C01786=1045.615,121.448,-88.791,170.522,36.741,156.917
C01787=1045.608,121.199,-88.770,170.520,36.740,156.916
C01788=1045.602,120.950,-88.750,170.518,36.739,156.916
C01789=1045.596,120.700,-88.729,170.516,36.737,156.916
C01790=1045.590,120.451,-88.709,170.514,36.736,156.916
C01791=1045.581,120.085,-88.679,170.511,36.733,156.915
C01792=1045.572,119.720,-88.649,170.509,36.731,156.915
C01793=1045.563,119.355,-88.619,170.505,36.729,156.914
C01794=1045.555,118.989,-88.589,170.503,36.726,156.914
C01795=1045.548,118.740,-88.568,170.501,36.725,156.914
C01796=1045.542,118.491,-88.548,170.499,36.723,156.913
C01797=1045.536,118.241,-88.528,170.498,36.722,156.913
C01798=1045.530,117.992,-88.508,170.495,36.721,156.913
C01799=1045.524,117.744,-88.488,170.493,36.719,156.912
C01800=1045.518,117.494,-88.467,170.491,36.718,156.912
C01801=1045.512,117.245,-88.447,170.490,36.716,156.912
C01802=1045.506,116.996,-88.427,170.488,36.715,156.911
C01803=1045.500,116.747,-88.406,170.486,36.713,156.911
C01804=1045.494,116.498,-88.385,170.483,36.711,156.911
C01805=1045.488,116.249,-88.365,170.482,36.710,156.911
C01806=1045.482,116.000,-88.345,170.480,36.708,156.910
C01807=1045.476,115.751,-88.324,170.478,36.707,156.910
C01808=1045.470,115.501,-88.304,170.477,36.705,156.910
C01809=1045.464,115.252,-88.284,170.474,36.703,156.909
C01810=1045.458,115.004,-88.264,170.472,36.702,156.909
C01811=1045.452,114.754,-88.243,170.471,36.700,156.909
C01812=1045.446,114.505,-88.223,170.469,36.699,156.908
C01813=1045.440,114.256,-88.203,170.467,36.698,156.908
C01814=1045.434,114.007,-88.183,170.464,36.696,156.908
C01815=1045.428,113.757,-88.162,170.463,36.695,156.908
C01816=1045.422,113.509,-88.142,170.461,36.693,156.907
C01817=1045.416,113.260,-88.122,170.459,36.692,156.907
C01818=1045.410,113.010,-88.102,170.458,36.690,156.907
C01819=1045.404,112.761,-88.082,170.456,36.689,156.906
C01820=1045.398,112.512,-88.063,170.453,36.687,156.906
C01821=1045.391,112.263,-88.043,170.451,36.686,156.906
C01822=1045.385,112.014,-88.023,170.450,36.684,156.906
C01823=1045.379,111.765,-88.003,170.448,36.683,156.905
C01824=1045.373,111.515,-87.982,170.446,36.681,156.905
C01825=1045.367,111.267,-87.962,170.444,36.680,156.905
C01826=1045.361,111.018,-87.942,170.442,36.679,156.904
C01827=1045.354,110.768,-87.922,170.440,36.677,156.904
C01828=1045.348,110.519,-87.903,170.438,36.676,156.904
C01829=1045.342,110.270,-87.883,170.437,36.674,156.904
C01830=1045.336,110.020,-87.863,170.435,36.673,156.903
C01831=1045.328,109.735,-87.840,170.432,36.671,156.903
C01832=1045.322,109.449,-87.817,170.430,36.669,156.903
C01833=1045.314,109.163,-87.795,170.428,36.668,156.902
C01834=1045.308,108.877,-87.772,170.426,36.666,156.902
C01835=1045.301,108.627,-87.752,170.424,36.665,156.902
C01836=1045.295,108.379,-87.732,170.423,36.664,156.902
C01837=1045.288,108.130,-87.713,170.420,36.662,156.901
C01838=1045.283,107.881,-87.693,170.418,36.661,156.901
C01839=1045.276,107.631,-87.673,170.416,36.659,156.901
C01840=1045.270,107.382,-87.653,170.415,36.658,156.900
C01841=1045.264,107.133,-87.634,170.413,36.656,156.900
C01842=1045.258,106.883,-87.613,170.411,36.655,156.900
C01843=1045.251,106.635,-87.594,170.409,36.653,156.900
C01844=1045.245,106.386,-87.575,170.407,36.652,156.899
C01845=1045.239,106.137,-87.555,170.405,36.651,156.899
C01846=1045.233,105.887,-87.534,170.403,36.650,156.899
C01847=1045.227,105.638,-87.515,170.402,36.648,156.898
C01848=1045.221,105.389,-87.495,170.399,36.646,156.898
C01849=1045.214,105.140,-87.476,170.397,36.645,156.898
C01850=1045.208,104.890,-87.456,170.396,36.643,156.898
C01851=1045.202,104.642,-87.436,170.394,36.642,156.897
C01852=1045.196,104.392,-87.417,170.392,36.641,156.897
C01853=1045.190,104.143,-87.397,170.391,36.639,156.897
C01854=1045.184,103.894,-87.377,170.388,36.638,156.896
C01855=1045.177,103.645,-87.358,170.386,36.637,156.896
C01856=1045.171,103.396,-87.338,170.384,36.635,156.896
C01857=1045.166,103.146,-87.319,170.383,36.633,156.896
C01858=1045.160,102.898,-87.299,170.381,36.632,156.895
C01859=1045.154,102.649,-87.279,170.379,36.630,156.895
C01860=1045.147,102.399,-87.259,170.377,36.629,156.895
C01861=1045.141,102.150,-87.240,170.375,36.628,156.895
C01862=1045.135,101.901,-87.221,170.373,36.626,156.894
C01863=1045.129,101.652,-87.201,170.372,36.625,156.894
C01864=1045.123,101.402,-87.182,170.370,36.624,156.894
C01865=1045.117,101.154,-87.162,170.368,36.622,156.893
C01866=1045.110,100.904,-87.143,170.366,36.620,156.893
C01867=1045.104,100.655,-87.123,170.364,36.619,156.893
C01868=1045.098,100.406,-87.103,170.362,36.618,156.893
C01869=1045.092,100.157,-87.084,170.360,36.616,156.892
C01870=1045.086,99.908,-87.065,170.359,36.615,156.892
C01871=1045.079,99.658,-87.044,170.357,36.614,156.892
C01872=1045.073,99.409,-87.026,170.354,36.612,156.892
C01873=1045.067,99.160,-87.007,170.353,36.611,156.891
C01874=1045.061,98.911,-86.987,170.351,36.609,156.891
C01875=1045.055,98.662,-86.968,170.349,36.608,156.891
C01876=1045.048,98.413,-86.949,170.348,36.607,156.890
C01877=1045.042,98.163,-86.929,170.346,36.605,156.890
C01878=1045.035,97.914,-86.910,170.343,36.604,156.890
C01879=1045.029,97.665,-86.890,170.341,36.602,156.890
C01880=1045.024,97.416,-86.871,170.340,36.601,156.889
C01881=1045.017,97.167,-86.852,170.338,36.600,156.889
C01882=1045.011,96.918,-86.833,170.336,36.599,156.889
C01883=1045.005,96.669,-86.814,170.335,36.597,156.889
C01884=1044.999,96.418,-86.794,170.332,36.596,156.888
C01885=1044.992,96.170,-86.775,170.330,36.594,156.888
C01886=1044.986,95.921,-86.756,170.329,36.593,156.888
C01887=1044.980,95.671,-86.737,170.327,36.591,156.887
C01888=1044.974,95.423,-86.717,170.325,36.590,156.887
C01889=1044.967,95.173,-86.698,170.324,36.589,156.887
C01890=1044.962,94.924,-86.679,170.321,36.587,156.887
C01891=1044.956,94.675,-86.660,170.319,36.586,156.886
C01892=1044.949,94.426,-86.641,170.318,36.584,156.886
C01893=1044.943,94.176,-86.621,170.316,36.583,156.886
C01894=1044.937,93.927,-86.602,170.314,36.582,156.886
C01895=1044.930,93.642,-86.580,170.312,36.580,156.885
C01896=1044.923,93.355,-86.559,170.309,36.579,156.885
C01897=1044.916,93.069,-86.536,170.307,36.577,156.885
C01898=1044.909,92.783,-86.514,170.305,36.575,156.884
C01899=1044.902,92.534,-86.495,170.304,36.574,156.884
C01900=1044.896,92.285,-86.475,170.302,36.572,156.884
C01901=1044.890,92.036,-86.457,170.300,36.571,156.884
C01902=1044.884,91.787,-86.438,170.298,36.569,156.883
C01903=1044.878,91.538,-86.419,170.296,36.568,156.883
C01904=1044.872,91.288,-86.400,170.294,36.567,156.883
C01905=1044.866,91.039,-86.381,170.293,36.566,156.883
C01906=1044.860,90.790,-86.361,170.291,36.564,156.882
C01907=1044.853,90.541,-86.342,170.289,36.562,156.882
C01908=1044.848,90.292,-86.323,170.287,36.561,156.882
C01909=1044.841,90.043,-86.305,170.285,36.560,156.881
C01910=1044.835,89.793,-86.286,170.283,36.559,156.881
C01911=1044.829,89.544,-86.267,170.282,36.557,156.881
C01912=1044.822,89.294,-86.248,170.280,36.556,156.881
C01913=1044.816,89.045,-86.229,170.278,36.554,156.880
C01914=1044.809,88.796,-86.210,170.276,36.553,156.880
C01915=1044.803,88.546,-86.191,170.274,36.552,156.880
C01916=1044.797,88.297,-86.172,170.272,36.551,156.880
C01917=1044.791,88.048,-86.154,170.271,36.549,156.879
C01918=1044.784,87.799,-86.135,170.269,36.548,156.879
C01919=1044.779,87.550,-86.116,170.267,36.546,156.879
C01920=1044.772,87.301,-86.097,170.265,36.545,156.879
C01921=1044.766,87.051,-86.079,170.263,36.544,156.878
C01922=1044.759,86.802,-86.060,170.261,36.543,156.878
C01923=1044.754,86.553,-86.041,170.259,36.541,156.878
C01924=1044.747,86.304,-86.022,170.258,36.540,156.878
C01925=1044.741,86.055,-86.003,170.256,36.538,156.877
C01926=1044.734,85.805,-85.985,170.254,36.537,156.877
C01927=1044.729,85.556,-85.966,170.252,36.536,156.877
C01928=1044.722,85.307,-85.947,170.250,36.534,156.877
C01929=1044.716,85.058,-85.928,170.248,36.533,156.876
C01930=1044.709,84.809,-85.910,170.247,36.532,156.876
C01931=1044.703,84.560,-85.891,170.245,36.530,156.876
C01932=1044.697,84.310,-85.872,170.243,36.529,156.876
C01933=1044.691,84.061,-85.853,170.242,36.528,156.875
C01934=1044.684,83.812,-85.834,170.239,36.526,156.875
C01935=1044.678,83.562,-85.816,170.237,36.525,156.875
C01936=1044.673,83.313,-85.797,170.236,36.524,156.875
C01937=1044.666,83.064,-85.779,170.234,36.522,156.874
C01938=1044.660,82.815,-85.760,170.232,36.521,156.874
C01939=1044.654,82.566,-85.742,170.231,36.519,156.874
C01940=1044.647,82.317,-85.723,170.228,36.518,156.873
C01941=1044.642,82.067,-85.704,170.226,36.517,156.873
C01942=1044.636,81.818,-85.686,170.225,36.516,156.873
C01943=1044.629,81.569,-85.667,170.223,36.514,156.873
C01944=1044.623,81.320,-85.649,170.221,36.513,156.872
C01945=1044.616,81.070,-85.630,170.220,36.511,156.872
C01946=1044.611,80.821,-85.611,170.218,36.510,156.872
C01947=1044.604,80.572,-85.592,170.215,36.509,156.872
C01948=1044.598,80.322,-85.574,170.214,36.507,156.871
C01949=1044.592,80.074,-85.556,170.212,36.506,156.871
C01950=1044.586,79.825,-85.537,170.210,36.504,156.871
C01951=1044.580,79.575,-85.518,170.209,36.503,156.871
C01952=1044.574,79.325,-85.500,170.207,36.502,156.870
C01953=1044.568,79.076,-85.481,170.204,36.500,156.870
C01954=1044.561,78.827,-85.463,170.203,36.499,156.870
C01955=1044.555,78.578,-85.444,170.201,36.497,156.870
C01956=1044.549,78.328,-85.426,170.199,36.496,156.869
C01957=1044.543,78.080,-85.408,170.198,36.495,156.869
C01958=1044.536,77.831,-85.389,170.196,36.494,156.869
C01959=1044.529,77.544,-85.368,170.194,36.492,156.869
C01960=1044.523,77.258,-85.347,170.191,36.491,156.868
C01961=1044.515,76.972,-85.326,170.189,36.489,156.868
C01962=1044.508,76.686,-85.304,170.187,36.487,156.868
C01963=1044.502,76.437,-85.286,170.186,36.486,156.867
C01964=1044.496,76.188,-85.268,170.184,36.485,156.867
C01965=1044.490,75.939,-85.249,170.182,36.484,156.867
C01966=1044.483,75.689,-85.232,170.180,36.482,156.867
C01967=1044.476,75.440,-85.213,170.178,36.481,156.866
C01968=1044.470,75.191,-85.195,170.176,36.479,156.866
C01969=1044.464,74.941,-85.177,170.174,36.478,156.866
C01970=1044.457,74.692,-85.158,170.173,36.477,156.866
C01971=1044.452,74.443,-85.141,170.171,36.476,156.865
C01972=1044.445,74.194,-85.122,170.169,36.474,156.865
C01973=1044.439,73.945,-85.103,170.167,36.473,156.865
C01974=1044.433,73.695,-85.085,170.165,36.472,156.865
C01975=1044.426,73.446,-85.067,170.163,36.471,156.864
C01976=1044.420,73.196,-85.049,170.162,36.469,156.864
C01977=1044.415,72.948,-85.031,170.160,36.467,156.864
C01978=1044.408,72.698,-85.013,170.158,36.466,156.864
C01979=1044.402,72.449,-84.994,170.157,36.465,156.863
C01980=1044.395,72.199,-84.977,170.154,36.464,156.863
C01981=1044.389,71.950,-84.958,170.152,36.462,156.863
C01982=1044.383,71.701,-84.940,170.151,36.461,156.863
C01983=1044.377,71.452,-84.922,170.149,36.460,156.862
C01984=1044.371,71.202,-84.904,170.147,36.459,156.862
C01985=1044.364,70.953,-84.885,170.146,36.457,156.862
C01986=1044.359,70.704,-84.868,170.143,36.455,156.862
C01987=1044.352,70.455,-84.849,170.141,36.454,156.861
C01988=1044.346,70.205,-84.831,170.140,36.453,156.861
C01989=1044.339,69.956,-84.814,170.138,36.452,156.861
C01990=1044.333,69.707,-84.795,170.136,36.450,156.861
C01991=1044.327,69.458,-84.777,170.135,36.449,156.860
C01992=1044.321,69.209,-84.759,170.133,36.448,156.860
C01993=1044.315,68.959,-84.741,170.130,36.447,156.860
C01994=1044.308,68.709,-84.724,170.129,36.445,156.860
C01995=1044.302,68.461,-84.705,170.127,36.444,156.860
C01996=1044.296,68.211,-84.687,170.125,36.443,156.859
C01997=1044.290,67.962,-84.669,170.124,36.442,156.859
C01998=1044.283,67.713,-84.651,170.122,36.440,156.859
C01999=1044.277,67.464,-84.634,170.120,36.438,156.858
C02000=1044.271,67.214,-84.616,170.117,36.437,156.858
C02001=1044.265,66.965,-84.597,170.116,36.436,156.858
C02002=1044.258,66.715,-84.580,170.114,36.435,156.858
C02003=1044.252,66.466,-84.562,170.112,36.433,156.857
C02004=1044.246,66.217,-84.544,170.111,36.432,156.857
C02005=1044.240,65.968,-84.526,170.109,36.431,156.857
C02006=1044.233,65.718,-84.508,170.107,36.430,156.857
C02007=1044.227,65.469,-84.491,170.105,36.428,156.857
C02008=1044.221,65.220,-84.472,170.103,36.427,156.856
C02009=1044.214,64.970,-84.455,170.101,36.426,156.856
C02010=1044.209,64.721,-84.437,170.100,36.425,156.856
C02011=1044.202,64.472,-84.419,170.098,36.423,156.856
C02012=1044.195,64.223,-84.401,170.096,36.422,156.855
C02013=1044.189,63.973,-84.383,170.095,36.421,156.855
C02014=1044.184,63.724,-84.366,170.093,36.420,156.855
C02015=1044.177,63.475,-84.348,170.090,36.418,156.855
C02016=1044.170,63.225,-84.331,170.088,36.417,156.854
C02017=1044.164,62.976,-84.313,170.087,36.416,156.854
C02018=1044.157,62.727,-84.295,170.085,36.415,156.854
C02019=1044.151,62.478,-84.278,170.083,36.413,156.854
C02020=1044.144,62.228,-84.260,170.082,36.412,156.853
C02021=1044.139,61.979,-84.243,170.080,36.411,156.853
C02022=1044.132,61.730,-84.225,170.078,36.410,156.853
C02023=1044.124,61.443,-84.205,170.075,36.408,156.853
C02024=1044.117,61.157,-84.185,170.073,36.407,156.853
C02025=1044.110,60.871,-84.165,170.071,36.406,156.852
C02026=1044.103,60.585,-84.145,170.069,36.404,156.852
C02027=1044.096,60.335,-84.127,170.068,36.403,156.852
C02028=1044.090,60.085,-84.110,170.066,36.402,156.852
C02029=1044.083,59.837,-84.092,170.063,36.401,156.851
C02030=1044.076,59.588,-84.074,170.062,36.399,156.851
C02031=1044.070,59.338,-84.057,170.060,36.398,156.851
C02032=1044.064,59.089,-84.040,170.058,36.397,156.851
C02033=1044.058,58.840,-84.022,170.056,36.396,156.850
C02034=1044.051,58.590,-84.004,170.055,36.394,156.850
C02035=1044.045,58.342,-83.987,170.053,36.393,156.850
C02036=1044.039,58.092,-83.969,170.051,36.392,156.850
C02037=1044.032,57.843,-83.952,170.049,36.391,156.849
C02038=1044.026,57.593,-83.934,170.047,36.389,156.849
C02039=1044.019,57.344,-83.917,170.045,36.388,156.849
C02040=1044.013,57.095,-83.900,170.043,36.387,156.849
C02041=1044.007,56.845,-83.882,170.042,36.386,156.849
C02042=1044.000,56.596,-83.865,170.040,36.385,156.848
C02043=1043.995,56.346,-83.848,170.038,36.384,156.848
C02044=1043.988,56.097,-83.831,170.037,36.382,156.848
C02045=1043.982,55.848,-83.814,170.034,36.381,156.848
C02046=1043.976,55.598,-83.796,170.032,36.380,156.848
C02047=1043.969,55.349,-83.778,170.031,36.379,156.847
C02048=1043.963,55.100,-83.761,170.029,36.377,156.847
C02049=1043.957,54.851,-83.744,170.027,36.376,156.847
C02050=1043.950,54.602,-83.727,170.025,36.375,156.847
C02051=1043.944,54.352,-83.709,170.024,36.373,156.846
C02052=1043.937,54.103,-83.691,170.021,36.372,156.846
C02053=1043.931,53.854,-83.674,170.019,36.371,156.846
C02054=1043.925,53.604,-83.657,170.018,36.370,156.846
C02055=1043.919,53.355,-83.640,170.016,36.368,156.845
C02056=1043.913,53.105,-83.622,170.014,36.367,156.845
C02057=1043.907,52.856,-83.605,170.012,36.366,156.845
C02058=1043.900,52.607,-83.588,170.011,36.365,156.845
C02059=1043.894,52.358,-83.570,170.009,36.363,156.844
C02060=1043.888,52.108,-83.554,170.006,36.362,156.844
C02061=1043.881,51.859,-83.537,170.005,36.361,156.844
C02062=1043.875,51.609,-83.519,170.003,36.360,156.844
C02063=1043.869,51.361,-83.502,170.001,36.358,156.844
C02064=1043.862,51.111,-83.485,170.000,36.357,156.843
C02065=1043.857,50.862,-83.468,169.998,36.356,156.843
C02066=1043.850,50.612,-83.450,169.996,36.355,156.843
C02067=1043.844,50.363,-83.433,169.993,36.353,156.843
C02068=1043.838,50.114,-83.415,169.992,36.352,156.842
C02069=1043.831,49.865,-83.398,169.990,36.351,156.842
C02070=1043.825,49.615,-83.382,169.988,36.349,156.842
C02071=1043.819,49.366,-83.364,169.987,36.348,156.842
C02072=1043.813,49.116,-83.347,169.985,36.347,156.841
C02073=1043.807,48.867,-83.329,169.983,36.346,156.841
C02074=1043.800,48.617,-83.313,169.981,36.344,156.841
C02075=1043.794,48.369,-83.296,169.979,36.343,156.841
C02076=1043.788,48.119,-83.278,169.977,36.342,156.840
C02077=1043.782,47.869,-83.262,169.975,36.341,156.840
C02078=1043.775,47.620,-83.244,169.974,36.339,156.840
C02079=1043.770,47.371,-83.227,169.972,36.338,156.840
C02080=1043.763,47.121,-83.210,169.970,36.337,156.840
C02081=1043.757,46.872,-83.193,169.969,36.336,156.839
C02082=1043.751,46.624,-83.176,169.966,36.334,156.839
C02083=1043.745,46.373,-83.159,169.964,36.333,156.839
C02084=1043.739,46.124,-83.142,169.963,36.332,156.839
C02085=1043.732,45.875,-83.125,169.961,36.330,156.838
C02086=1043.727,45.625,-83.108,169.959,36.329,156.838
C02087=1043.720,45.339,-83.088,169.957,36.328,156.838
C02088=1043.712,45.052,-83.068,169.955,36.326,156.838
C02089=1043.705,44.766,-83.050,169.952,36.325,156.837
C02090=1043.698,44.480,-83.030,169.950,36.323,156.837
C02091=1043.692,44.230,-83.012,169.949,36.322,156.837
C02092=1043.686,43.981,-82.995,169.947,36.321,156.837
C02093=1043.679,43.731,-82.978,169.945,36.320,156.836
C02094=1043.674,43.482,-82.961,169.944,36.318,156.836
C02095=1043.668,43.233,-82.944,169.942,36.317,156.836
C02096=1043.661,42.983,-82.928,169.940,36.316,156.836
C02097=1043.655,42.734,-82.911,169.937,36.315,156.835
C02098=1043.648,42.484,-82.894,169.936,36.313,156.835
C02099=1043.642,42.235,-82.877,169.934,36.312,156.835
C02100=1043.636,41.986,-82.861,169.932,36.311,156.835
C02101=1043.629,41.737,-82.843,169.930,36.309,156.835
C02102=1043.623,41.487,-82.827,169.929,36.308,156.834
C02103=1043.616,41.238,-82.810,169.927,36.307,156.834
C02104=1043.610,40.989,-82.794,169.925,36.306,156.834
C02105=1043.604,40.739,-82.777,169.923,36.305,156.834
C02106=1043.598,40.490,-82.760,169.921,36.304,156.833
C02107=1043.592,40.240,-82.744,169.919,36.302,156.833
C02108=1043.586,39.991,-82.726,169.917,36.301,156.833
C02109=1043.580,39.741,-82.710,169.916,36.300,156.833
C02110=1043.573,39.493,-82.693,169.914,36.299,156.833
C02111=1043.567,39.243,-82.676,169.912,36.297,156.832
C02112=1043.561,38.993,-82.660,169.909,36.296,156.832
C02113=1043.555,38.744,-82.643,169.908,36.295,156.832
C02114=1043.549,38.495,-82.626,169.906,36.294,156.832
C02115=1043.542,38.245,-82.610,169.904,36.293,156.832
C02116=1043.536,37.996,-82.593,169.903,36.292,156.831
C02117=1043.530,37.747,-82.577,169.901,36.290,156.831
C02118=1043.523,37.497,-82.560,169.899,36.289,156.831
C02119=1043.517,37.248,-82.543,169.897,36.288,156.831
C02120=1043.510,36.998,-82.526,169.896,36.287,156.830
C02121=1043.505,36.749,-82.510,169.893,36.285,156.830
C02122=1043.498,36.500,-82.494,169.891,36.285,156.830
C02123=1043.491,36.250,-82.477,169.889,36.283,156.830
C02124=1043.485,36.001,-82.461,169.888,36.282,156.830
C02125=1043.479,35.752,-82.445,169.886,36.281,156.829
C02126=1043.472,35.502,-82.427,169.884,36.280,156.829
C02127=1043.466,35.253,-82.411,169.882,36.279,156.829
C02128=1043.460,35.004,-82.395,169.880,36.278,156.829
C02129=1043.453,34.754,-82.379,169.878,36.276,156.829
C02130=1043.447,34.504,-82.362,169.876,36.275,156.828
C02131=1043.441,34.256,-82.346,169.874,36.274,156.828
C02132=1043.435,34.006,-82.329,169.872,36.273,156.828
C02133=1043.428,33.757,-82.313,169.871,36.272,156.828
C02134=1043.422,33.507,-82.297,169.869,36.271,156.827
C02135=1043.416,33.258,-82.281,169.867,36.269,156.827
C02136=1043.409,33.009,-82.263,169.865,36.268,156.827
C02137=1043.403,32.759,-82.247,169.864,36.267,156.827
C02138=1043.397,32.510,-82.231,169.861,36.266,156.827
C02139=1043.390,32.261,-82.215,169.859,36.265,156.826
C02140=1043.384,32.011,-82.199,169.857,36.264,156.826
C02141=1043.378,31.761,-82.182,169.856,36.262,156.826
C02142=1043.371,31.513,-82.165,169.854,36.261,156.826
C02143=1043.365,31.263,-82.149,169.852,36.260,156.825
C02144=1043.358,31.014,-82.133,169.850,36.259,156.825
C02145=1043.352,30.764,-82.117,169.849,36.258,156.825
C02146=1043.346,30.515,-82.101,169.846,36.257,156.825
C02147=1043.340,30.266,-82.084,169.844,36.255,156.825
C02148=1043.334,30.015,-82.068,169.842,36.254,156.824
C02149=1043.327,29.766,-82.052,169.840,36.253,156.824
C02150=1043.321,29.517,-82.036,169.839,36.252,156.824
C02151=1043.314,29.231,-82.017,169.837,36.251,156.824
C02152=1043.307,28.944,-81.998,169.835,36.249,156.824
C02153=1043.300,28.657,-81.980,169.833,36.248,156.823
C02154=1043.292,28.370,-81.961,169.830,36.246,156.823
C02155=1043.286,28.121,-81.945,169.828,36.245,156.823
C02156=1043.279,27.872,-81.929,169.826,36.244,156.823
C02157=1043.273,27.623,-81.913,169.824,36.243,156.823
C02158=1043.267,27.373,-81.897,169.822,36.242,156.822
C02159=1043.260,27.124,-81.880,169.821,36.241,156.822
C02160=1043.254,26.874,-81.864,169.819,36.240,156.822
C02161=1043.248,26.625,-81.848,169.817,36.239,156.822
C02162=1043.242,26.376,-81.832,169.815,36.237,156.821
C02163=1043.236,26.127,-81.816,169.813,36.236,156.821
C02164=1043.228,25.877,-81.800,169.811,36.236,156.821
C02165=1043.222,25.627,-81.784,169.809,36.234,156.821
C02166=1043.216,25.378,-81.768,169.807,36.233,156.821
C02167=1043.210,25.128,-81.753,169.805,36.232,156.821
C02168=1043.204,24.879,-81.736,169.804,36.231,156.820
C02169=1043.197,24.629,-81.720,169.802,36.230,156.820
C02170=1043.191,24.380,-81.704,169.800,36.228,156.820
C02171=1043.184,24.131,-81.688,169.798,36.228,156.820
C02172=1043.178,23.882,-81.672,169.795,36.227,156.820
C02173=1043.172,23.632,-81.656,169.794,36.225,156.819
C02174=1043.166,23.383,-81.641,169.792,36.224,156.819
C02175=1043.159,23.133,-81.624,169.790,36.223,156.819
C02176=1043.153,22.884,-81.609,169.788,36.222,156.819
C02177=1043.147,22.634,-81.592,169.786,36.221,156.818
C02178=1043.140,22.385,-81.577,169.785,36.219,156.818
C02179=1043.134,22.136,-81.560,169.783,36.219,156.818
C02180=1043.128,21.886,-81.546,169.781,36.218,156.818
C02181=1043.122,21.637,-81.529,169.778,36.216,156.818
C02182=1043.115,21.388,-81.514,169.776,36.215,156.817
C02183=1043.109,21.138,-81.497,169.775,36.214,156.817
C02184=1043.103,20.888,-81.481,169.773,36.213,156.817
C02185=1043.096,20.639,-81.466,169.771,36.212,156.817
C02186=1043.090,20.389,-81.450,169.769,36.211,156.817
C02187=1043.084,20.140,-81.434,169.767,36.210,156.817
C02188=1043.078,19.890,-81.418,169.766,36.209,156.816
C02189=1043.071,19.641,-81.403,169.764,36.207,156.816
C02190=1043.065,19.392,-81.386,169.762,36.207,156.816
C02191=1043.059,19.143,-81.371,169.759,36.205,156.816
C02192=1043.052,18.893,-81.356,169.757,36.204,156.815
C02193=1043.046,18.644,-81.340,169.755,36.203,156.815
C02194=1043.039,18.394,-81.323,169.754,36.202,156.815
C02195=1043.033,18.144,-81.308,169.752,36.201,156.815
C02196=1043.027,17.895,-81.292,169.750,36.200,156.815
C02197=1043.020,17.646,-81.277,169.748,36.199,156.815
C02198=1043.014,17.396,-81.261,169.746,36.198,156.814
C02199=1043.008,17.147,-81.245,169.745,36.197,156.814
C02200=1043.002,16.897,-81.230,169.742,36.196,156.814
C02201=1042.995,16.648,-81.214,169.740,36.194,156.814
C02202=1042.989,16.399,-81.199,169.738,36.194,156.814
C02203=1042.983,16.149,-81.183,169.736,36.193,156.813
C02204=1042.976,15.900,-81.167,169.734,36.191,156.813
C02205=1042.970,15.650,-81.152,169.733,36.190,156.813
C02206=1042.964,15.401,-81.136,169.731,36.189,156.813
C02207=1042.957,15.152,-81.120,169.729,36.188,156.813
C02208=1042.952,14.902,-81.105,169.727,36.187,156.812
C02209=1042.945,14.653,-81.089,169.725,36.186,156.812
C02210=1042.938,14.403,-81.074,169.722,36.185,156.812
C02211=1042.933,14.154,-81.058,169.721,36.184,156.812
C02212=1042.926,13.904,-81.043,169.719,36.183,156.812
C02213=1042.919,13.655,-81.027,169.717,36.182,156.811
C02214=1042.913,13.406,-81.013,169.715,36.181,156.811
C02215=1042.906,13.120,-80.995,169.713,36.180,156.811
C02216=1042.898,12.835,-80.977,169.711,36.178,156.811
C02217=1042.891,12.550,-80.959,169.709,36.177,156.811
C02218=1042.884,12.265,-80.941,169.707,36.176,156.811
C02219=1042.877,12.015,-80.926,169.704,36.175,156.810
C02220=1042.871,11.765,-80.911,169.702,36.174,156.810
C02221=1042.864,11.516,-80.896,169.700,36.173,156.810
C02222=1042.858,11.267,-80.881,169.698,36.172,156.810
C02223=1042.851,11.017,-80.865,169.696,36.171,156.810
C02224=1042.845,10.768,-80.850,169.694,36.170,156.809
C02225=1042.839,10.518,-80.835,169.692,36.169,156.809
C02226=1042.832,10.269,-80.819,169.691,36.168,156.809
C02227=1042.826,10.019,-80.804,169.689,36.167,156.809
C02228=1042.819,9.770,-80.788,169.687,36.166,156.809
C02229=1042.813,9.520,-80.773,169.685,36.165,156.809
C02230=1042.807,9.271,-80.758,169.682,36.164,156.808
C02231=1042.800,9.022,-80.743,169.680,36.163,156.808
C02232=1042.793,8.772,-80.728,169.678,36.162,156.808
C02233=1042.788,8.522,-80.712,169.676,36.161,156.808
C02234=1042.781,8.273,-80.697,169.675,36.160,156.808
C02235=1042.775,8.023,-80.682,169.673,36.159,156.808
C02236=1042.768,7.774,-80.667,169.671,36.158,156.807
C02237=1042.762,7.524,-80.652,169.669,36.157,156.807
C02238=1042.755,7.275,-80.636,169.667,36.156,156.807
C02239=1042.750,7.026,-80.622,169.665,36.155,156.807
C02240=1042.743,6.776,-80.607,169.662,36.154,156.807
C02241=1042.736,6.527,-80.591,169.660,36.153,156.807
C02242=1042.730,6.278,-80.576,169.659,36.152,156.806
C02243=1042.724,6.028,-80.560,169.657,36.151,156.806
C02244=1042.718,5.778,-80.545,169.655,36.150,156.806
C02245=1042.712,5.528,-80.531,169.653,36.149,156.806
C02246=1042.705,5.279,-80.515,169.651,36.148,156.806
C02247=1042.699,5.030,-80.500,169.649,36.147,156.805
C02248=1042.693,4.781,-80.485,169.647,36.146,156.805
C02249=1042.686,4.531,-80.470,169.645,36.145,156.805
C02250=1042.680,4.282,-80.455,169.643,36.144,156.805
C02251=1042.673,4.033,-80.440,169.641,36.143,156.805
C02252=1042.667,3.783,-80.425,169.639,36.142,156.805
C02253=1042.661,3.533,-80.410,169.637,36.141,156.804
C02254=1042.655,3.283,-80.394,169.635,36.140,156.804
C02255=1042.649,3.034,-80.380,169.633,36.139,156.804
C02256=1042.642,2.785,-80.364,169.631,36.138,156.804
C02257=1042.636,2.536,-80.349,169.629,36.137,156.804
C02258=1042.630,2.286,-80.334,169.627,36.136,156.803
C02259=1042.623,2.036,-80.319,169.625,36.135,156.803
C02260=1042.617,1.787,-80.304,169.624,36.134,156.803
C02261=1042.611,1.538,-80.290,169.622,36.133,156.803
C02262=1042.605,1.288,-80.275,169.619,36.132,156.803
C02263=1042.598,1.038,-80.260,169.617,36.131,156.803
C02264=1042.592,0.789,-80.245,169.615,36.130,156.802
C02265=1042.585,0.540,-80.229,169.613,36.129,156.802
C02266=1042.580,0.291,-80.215,169.611,36.128,156.802
C02267=1042.573,0.041,-80.200,169.609,36.127,156.802
C02268=1042.567,-0.209,-80.185,169.607,36.126,156.802
C02269=1042.560,-0.458,-80.170,169.605,36.125,156.802
C02270=1042.555,-0.707,-80.155,169.604,36.124,156.801
C02271=1042.548,-0.957,-80.140,169.602,36.123,156.801
C02272=1042.543,-1.207,-80.125,169.599,36.121,156.801
C02273=1042.536,-1.457,-80.110,169.597,36.121,156.801
C02274=1042.530,-1.705,-80.095,169.595,36.120,156.801
C02275=1042.524,-1.955,-80.080,169.593,36.119,156.801
C02276=1042.518,-2.205,-80.065,169.591,36.118,156.800
C02277=1042.511,-2.454,-80.050,169.589,36.117,156.800
C02278=1042.505,-2.703,-80.036,169.587,36.116,156.800
C02279=1042.498,-2.987,-80.019,169.585,36.114,156.800
C02280=1042.490,-3.270,-80.002,169.583,36.113,156.799
C02281=1042.484,-3.554,-79.985,169.581,36.112,156.799
C02282=1042.477,-3.838,-79.969,169.578,36.111,156.799
C02283=1042.470,-4.087,-79.954,169.576,36.110,156.799
C02284=1042.464,-4.336,-79.940,169.574,36.109,156.799
C02285=1042.458,-4.586,-79.925,169.572,36.108,156.799
C02286=1042.451,-4.835,-79.910,169.570,36.108,156.799
C02287=1042.444,-5.085,-79.896,169.568,36.106,156.798
C02288=1042.439,-5.334,-79.882,169.566,36.106,156.798
C02289=1042.432,-5.584,-79.867,169.564,36.105,156.798
C02290=1042.425,-5.833,-79.852,169.562,36.104,156.798
C02291=1042.419,-6.083,-79.837,169.560,36.103,156.798
C02292=1042.413,-6.332,-79.823,169.558,36.102,156.798
C02293=1042.407,-6.582,-79.808,169.556,36.101,156.797
C02294=1042.400,-6.831,-79.794,169.554,36.101,156.797
C02295=1042.393,-7.081,-79.779,169.551,36.099,156.797
C02296=1042.388,-7.330,-79.765,169.549,36.099,156.797
C02297=1042.381,-7.579,-79.750,169.547,36.097,156.797
C02298=1042.375,-7.830,-79.736,169.545,36.097,156.797
C02299=1042.369,-8.079,-79.722,169.543,36.096,156.797
C02300=1042.362,-8.328,-79.707,169.541,36.095,156.796
C02301=1042.355,-8.578,-79.692,169.539,36.094,156.796
C02302=1042.350,-8.827,-79.678,169.537,36.093,156.796
C02303=1042.343,-9.077,-79.663,169.535,36.092,156.796
C02304=1042.336,-9.326,-79.649,169.533,36.091,156.796
C02305=1042.330,-9.575,-79.635,169.531,36.090,156.796
C02306=1042.324,-9.825,-79.620,169.530,36.090,156.795
C02307=1042.317,-10.075,-79.606,169.527,36.089,156.795
C02308=1042.311,-10.324,-79.591,169.525,36.088,156.795
C02309=1042.305,-10.574,-79.577,169.523,36.087,156.795
C02310=1042.298,-10.823,-79.563,169.521,36.086,156.795
C02311=1042.292,-11.072,-79.548,169.519,36.085,156.795
C02312=1042.286,-11.323,-79.534,169.517,36.084,156.795
C02313=1042.280,-11.571,-79.520,169.515,36.083,156.794
C02314=1042.274,-11.821,-79.505,169.513,36.082,156.794
C02315=1042.267,-12.071,-79.491,169.511,36.082,156.794
C02316=1042.261,-12.320,-79.477,169.509,36.080,156.794
C02317=1042.255,-12.570,-79.463,169.507,36.080,156.794
C02318=1042.248,-12.820,-79.448,169.505,36.079,156.794
C02319=1042.242,-13.068,-79.434,169.502,36.078,156.793
C02320=1042.236,-13.319,-79.419,169.500,36.077,156.793
C02321=1042.230,-13.568,-79.405,169.498,36.076,156.793
C02322=1042.223,-13.818,-79.391,169.496,36.075,156.793
C02323=1042.217,-14.067,-79.377,169.494,36.074,156.793
C02324=1042.211,-14.317,-79.362,169.492,36.073,156.793
C02325=1042.204,-14.566,-79.348,169.490,36.073,156.793
C02326=1042.199,-14.815,-79.334,169.488,36.072,156.792
C02327=1042.192,-15.065,-79.319,169.486,36.071,156.792
C02328=1042.186,-15.314,-79.305,169.484,36.070,156.792
C02329=1042.180,-15.564,-79.291,169.482,36.069,156.792
C02330=1042.173,-15.813,-79.277,169.480,36.068,156.792
C02331=1042.167,-16.063,-79.263,169.478,36.067,156.792
C02332=1042.160,-16.313,-79.249,169.476,36.067,156.792
C02333=1042.155,-16.562,-79.235,169.473,36.066,156.791
C02334=1042.148,-16.812,-79.221,169.471,36.065,156.791
C02335=1042.141,-17.061,-79.207,169.469,36.064,156.791
C02336=1042.135,-17.311,-79.193,169.467,36.063,156.791
C02337=1042.129,-17.560,-79.179,169.465,36.063,156.791
C02338=1042.123,-17.810,-79.165,169.463,36.062,156.791
C02339=1042.116,-18.060,-79.151,169.461,36.061,156.791
C02340=1042.109,-18.309,-79.137,169.459,36.060,156.790
C02341=1042.103,-18.559,-79.123,169.457,36.059,156.790
C02342=1042.097,-18.808,-79.109,169.455,36.059,156.790
C02343=1042.089,-19.090,-79.093,169.452,36.057,156.790
C02344=1042.083,-19.371,-79.078,169.450,36.057,156.790
C02345=1042.075,-19.654,-79.062,169.448,36.056,156.790
C02346=1042.069,-19.936,-79.046,169.444,36.055,156.790
C02347=1042.062,-20.185,-79.032,169.442,36.054,156.789
C02348=1042.055,-20.434,-79.018,169.440,36.053,156.789
C02349=1042.050,-20.684,-79.004,169.438,36.053,156.789
C02350=1042.043,-20.934,-78.990,169.436,36.051,156.789
C02351=1042.036,-21.182,-78.976,169.434,36.051,156.789
C02352=1042.030,-21.433,-78.962,169.432,36.050,156.789
C02353=1042.024,-21.682,-78.949,169.430,36.049,156.789
C02354=1042.018,-21.932,-78.934,169.428,36.049,156.789
C02355=1042.012,-22.181,-78.921,169.426,36.048,156.788
C02356=1042.005,-22.430,-78.907,169.424,36.047,156.788
C02357=1041.999,-22.680,-78.893,169.422,36.046,156.788
C02358=1041.993,-22.929,-78.879,169.420,36.046,156.788
C02359=1041.987,-23.179,-78.865,169.418,36.045,156.788
C02360=1041.980,-23.429,-78.852,169.416,36.044,156.788
C02361=1041.974,-23.679,-78.838,169.413,36.043,156.788
C02362=1041.968,-23.928,-78.824,169.411,36.042,156.788
C02363=1041.962,-24.177,-78.810,169.409,36.042,156.787
C02364=1041.955,-24.427,-78.797,169.407,36.041,156.787
C02365=1041.949,-24.676,-78.783,169.404,36.040,156.787
C02366=1041.942,-24.926,-78.769,169.402,36.039,156.787
C02367=1041.936,-25.176,-78.756,169.400,36.038,156.787
C02368=1041.930,-25.425,-78.741,169.398,36.038,156.787
C02369=1041.924,-25.675,-78.728,169.396,36.036,156.787
C02370=1041.918,-25.924,-78.714,169.394,36.036,156.786
C02371=1041.911,-26.174,-78.700,169.392,36.035,156.786
C02372=1041.905,-26.423,-78.687,169.390,36.034,156.786
C02373=1041.900,-26.673,-78.673,169.388,36.034,156.786
C02374=1041.893,-26.923,-78.659,169.386,36.032,156.786
C02375=1041.887,-27.172,-78.646,169.383,36.032,156.786
C02376=1041.880,-27.422,-78.632,169.381,36.031,156.786
C02377=1041.873,-27.671,-78.618,169.379,36.030,156.786
C02378=1041.867,-27.920,-78.605,169.377,36.030,156.785
C02379=1041.861,-28.170,-78.591,169.374,36.029,156.785
C02380=1041.855,-28.420,-78.578,169.372,36.028,156.785
C02381=1041.849,-28.669,-78.564,169.370,36.028,156.785
C02382=1041.842,-28.919,-78.551,169.368,36.027,156.785
C02383=1041.836,-29.168,-78.537,169.366,36.026,156.785
C02384=1041.829,-29.418,-78.524,169.364,36.026,156.785
C02385=1041.823,-29.667,-78.511,169.362,36.025,156.785
C02386=1041.816,-29.917,-78.497,169.360,36.024,156.785
C02387=1041.810,-30.166,-78.484,169.358,36.024,156.784
C02388=1041.804,-30.416,-78.470,169.355,36.023,156.784
C02389=1041.798,-30.666,-78.457,169.353,36.022,156.784
C02390=1041.791,-30.916,-78.444,169.351,36.022,156.784
C02391=1041.785,-31.165,-78.430,169.349,36.021,156.784
C02392=1041.779,-31.414,-78.417,169.347,36.020,156.784
C02393=1041.772,-31.664,-78.403,169.344,36.020,156.784
C02394=1041.766,-31.914,-78.390,169.342,36.019,156.784
C02395=1041.760,-32.163,-78.377,169.340,36.018,156.784
C02396=1041.753,-32.413,-78.363,169.338,36.018,156.783
C02397=1041.747,-32.662,-78.350,169.335,36.017,156.783
C02398=1041.740,-32.911,-78.337,169.333,36.016,156.783
C02399=1041.734,-33.161,-78.323,169.331,36.015,156.783
C02400=1041.728,-33.412,-78.310,169.329,36.014,156.783
C02401=1041.722,-33.661,-78.297,169.327,36.014,156.783
C02402=1041.716,-33.910,-78.283,169.325,36.013,156.783
C02403=1041.709,-34.160,-78.270,169.323,36.012,156.783
C02404=1041.703,-34.409,-78.257,169.321,36.012,156.782
C02405=1041.697,-34.659,-78.243,169.318,36.011,156.782
C02406=1041.691,-34.909,-78.231,169.316,36.010,156.782
C02407=1041.683,-35.189,-78.216,169.314,36.010,156.782
C02408=1041.677,-35.471,-78.201,169.312,36.009,156.782
C02409=1041.669,-35.751,-78.186,169.309,36.008,156.782
C02410=1041.663,-36.033,-78.171,169.306,36.008,156.782
C02411=1041.657,-36.282,-78.157,169.304,36.007,156.782
C02412=1041.650,-36.531,-78.144,169.301,36.006,156.782
C02413=1041.644,-36.781,-78.131,169.299,36.006,156.782
C02414=1041.637,-37.031,-78.117,169.297,36.005,156.781
C02415=1041.632,-37.280,-78.105,169.295,36.004,156.781
C02416=1041.625,-37.530,-78.091,169.293,36.004,156.781
C02417=1041.619,-37.779,-78.078,169.291,36.003,156.781
C02418=1041.613,-38.030,-78.065,169.289,36.002,156.781
C02419=1041.606,-38.279,-78.052,169.287,36.002,156.781
C02420=1041.600,-38.528,-78.039,169.284,36.001,156.781
C02421=1041.594,-38.778,-78.026,169.282,36.000,156.781
C02422=1041.588,-39.027,-78.013,169.280,36.000,156.781
C02423=1041.581,-39.277,-77.999,169.278,35.999,156.780
C02424=1041.575,-39.527,-77.987,169.276,35.998,156.780
C02425=1041.568,-39.776,-77.974,169.274,35.998,156.780
C02426=1041.562,-40.025,-77.961,169.271,35.997,156.780
C02427=1041.556,-40.275,-77.948,169.269,35.997,156.780
C02428=1041.549,-40.525,-77.935,169.267,35.996,156.780
C02429=1041.543,-40.775,-77.923,169.265,35.996,156.780
C02430=1041.537,-41.024,-77.909,169.262,35.995,156.780
C02431=1041.530,-41.273,-77.896,169.259,35.994,156.780
C02432=1041.524,-41.523,-77.884,169.257,35.994,156.780
C02433=1041.518,-41.772,-77.870,169.255,35.993,156.780
C02434=1041.511,-42.023,-77.858,169.253,35.993,156.780
C02435=1041.505,-42.272,-77.845,169.251,35.992,156.779
C02436=1041.499,-42.522,-77.832,169.249,35.991,156.779
C02437=1041.493,-42.771,-77.819,169.246,35.991,156.779
C02438=1041.487,-43.021,-77.806,169.244,35.990,156.779
C02439=1041.480,-43.270,-77.794,169.242,35.990,156.779
C02440=1041.474,-43.520,-77.781,169.240,35.989,156.779
C02441=1041.468,-43.769,-77.768,169.238,35.989,156.779
C02442=1041.461,-44.020,-77.755,169.235,35.988,156.779
C02443=1041.455,-44.269,-77.742,169.233,35.987,156.779
C02444=1041.448,-44.519,-77.730,169.231,35.987,156.779
C02445=1041.442,-44.768,-77.716,169.229,35.987,156.779
C02446=1041.436,-45.018,-77.704,169.227,35.986,156.778
C02447=1041.430,-45.267,-77.691,169.224,35.985,156.778
C02448=1041.423,-45.516,-77.679,169.222,35.985,156.778
C02449=1041.417,-45.766,-77.666,169.220,35.984,156.778
C02450=1041.411,-46.016,-77.653,169.218,35.983,156.778
C02451=1041.405,-46.266,-77.640,169.216,35.983,156.778
C02452=1041.398,-46.514,-77.628,169.213,35.983,156.778
C02453=1041.392,-46.764,-77.615,169.210,35.982,156.778
C02454=1041.386,-47.014,-77.602,169.208,35.981,156.778
C02455=1041.380,-47.264,-77.589,169.206,35.981,156.778
C02456=1041.374,-47.513,-77.577,169.204,35.981,156.778
C02457=1041.368,-47.763,-77.565,169.201,35.980,156.778
C02458=1041.361,-48.013,-77.551,169.199,35.979,156.777
C02459=1041.355,-48.263,-77.538,169.197,35.979,156.777
C02460=1041.348,-48.512,-77.526,169.195,35.978,156.777
C02461=1041.342,-48.762,-77.513,169.193,35.978,156.777
C02462=1041.336,-49.012,-77.501,169.190,35.977,156.777
C02463=1041.330,-49.261,-77.488,169.188,35.977,156.777
C02464=1041.323,-49.510,-77.475,169.186,35.976,156.777
C02465=1041.318,-49.760,-77.463,169.184,35.975,156.777
C02466=1041.312,-50.009,-77.451,169.181,35.975,156.777
C02467=1041.306,-50.259,-77.437,169.179,35.974,156.777
C02468=1041.299,-50.508,-77.425,169.177,35.974,156.777
C02469=1041.293,-50.759,-77.413,169.175,35.974,156.777
C02470=1041.286,-51.008,-77.401,169.173,35.973,156.776
C02471=1041.279,-51.289,-77.387,169.170,35.972,156.776
C02472=1041.272,-51.571,-77.373,169.167,35.972,156.776
C02473=1041.264,-51.852,-77.359,169.165,35.972,156.776
C02474=1041.257,-52.134,-77.345,169.162,35.971,156.776
C02475=1041.251,-52.384,-77.332,169.160,35.971,156.776
C02476=1041.244,-52.633,-77.320,169.158,35.970,156.776
C02477=1041.238,-52.883,-77.308,169.155,35.970,156.776
C02478=1041.232,-53.133,-77.296,169.153,35.970,156.776
C02479=1041.225,-53.382,-77.284,169.151,35.970,156.776
C02480=1041.219,-53.632,-77.271,169.148,35.969,156.776
C02481=1041.213,-53.882,-77.259,169.145,35.969,156.776
C02482=1041.206,-54.131,-77.247,169.143,35.968,156.776
C02483=1041.200,-54.381,-77.235,169.141,35.968,156.776
C02484=1041.194,-54.630,-77.223,169.139,35.967,156.776
C02485=1041.187,-54.880,-77.211,169.136,35.967,156.776
C02486=1041.181,-55.129,-77.198,169.134,35.967,156.776
C02487=1041.174,-55.378,-77.186,169.132,35.966,156.775
C02488=1041.169,-55.628,-77.173,169.129,35.966,156.775
C02489=1041.162,-55.878,-77.161,169.127,35.965,156.775
C02490=1041.155,-56.127,-77.149,169.125,35.965,156.775
C02491=1041.149,-56.377,-77.137,169.123,35.965,156.775
C02492=1041.143,-56.627,-77.125,169.120,35.965,156.775
C02493=1041.136,-56.876,-77.113,169.118,35.964,156.775
C02494=1041.130,-57.126,-77.100,169.116,35.964,156.775
C02495=1041.123,-57.376,-77.088,169.113,35.963,156.775
C02496=1041.117,-57.625,-77.076,169.111,35.963,156.775
C02497=1041.112,-57.875,-77.064,169.109,35.963,156.775
C02498=1041.105,-58.124,-77.052,169.107,35.963,156.775
C02499=1041.099,-58.374,-77.041,169.104,35.962,156.775
C02500=1041.093,-58.624,-77.028,169.102,35.962,156.775
C02501=1041.086,-58.874,-77.016,169.100,35.961,156.775
C02502=1041.079,-59.123,-77.004,169.097,35.961,156.775
C02503=1041.073,-59.373,-76.992,169.095,35.960,156.775
C02504=1041.067,-59.623,-76.980,169.093,35.960,156.775
C02505=1041.061,-59.872,-76.968,169.090,35.960,156.775
C02506=1041.055,-60.122,-76.956,169.088,35.960,156.775
C02507=1041.048,-60.371,-76.944,169.086,35.959,156.774
C02508=1041.042,-60.621,-76.932,169.084,35.959,156.775
C02509=1041.036,-60.871,-76.920,169.081,35.958,156.774
C02510=1041.030,-61.120,-76.908,169.079,35.958,156.774
C02511=1041.023,-61.370,-76.897,169.077,35.958,156.774
C02512=1041.017,-61.620,-76.884,169.074,35.958,156.774
C02513=1041.011,-61.869,-76.872,169.072,35.957,156.774
C02514=1041.004,-62.119,-76.860,169.070,35.957,156.774
C02515=1040.999,-62.369,-76.849,169.067,35.957,156.774
C02516=1040.992,-62.618,-76.837,169.065,35.956,156.774
C02517=1040.986,-62.868,-76.825,169.063,35.956,156.774
C02518=1040.980,-63.118,-76.812,169.060,35.955,156.774
C02519=1040.973,-63.367,-76.800,169.058,35.955,156.774
C02520=1040.967,-63.617,-76.789,169.056,35.955,156.774
C02521=1040.961,-63.866,-76.777,169.054,35.955,156.774
C02522=1040.955,-64.116,-76.765,169.050,35.954,156.774
C02523=1040.948,-64.366,-76.753,169.048,35.954,156.774
C02524=1040.943,-64.615,-76.742,169.046,35.953,156.774
C02525=1040.937,-64.865,-76.729,169.043,35.953,156.774
C02526=1040.930,-65.115,-76.717,169.041,35.953,156.774
C02527=1040.924,-65.363,-76.706,169.039,35.953,156.774
C02528=1040.918,-65.614,-76.695,169.036,35.952,156.774
C02529=1040.912,-65.864,-76.682,169.034,35.952,156.774
C02530=1040.905,-66.113,-76.670,169.032,35.952,156.774
C02531=1040.899,-66.363,-76.659,169.029,35.951,156.773
C02532=1040.893,-66.613,-76.647,169.027,35.951,156.773
C02533=1040.887,-66.862,-76.635,169.025,35.950,156.773
C02534=1040.881,-67.112,-76.624,169.022,35.950,156.773
C02535=1040.873,-67.394,-76.610,169.020,35.950,156.773
C02536=1040.867,-67.677,-76.597,169.017,35.950,156.773
C02537=1040.860,-67.960,-76.584,169.014,35.950,156.773
C02538=1040.853,-68.242,-76.571,169.012,35.949,156.773
C02539=1040.846,-68.492,-76.559,169.009,35.949,156.773
C02540=1040.841,-68.742,-76.547,169.007,35.948,156.773
C02541=1040.835,-68.991,-76.535,169.005,35.948,156.773
C02542=1040.828,-69.241,-76.523,169.002,35.947,156.773
C02543=1040.822,-69.491,-76.512,169.000,35.947,156.773
C02544=1040.817,-69.740,-76.500,168.998,35.947,156.773
C02545=1040.810,-69.990,-76.489,168.995,35.947,156.773
C02546=1040.804,-70.239,-76.477,168.993,35.947,156.773
C02547=1040.798,-70.490,-76.466,168.991,35.946,156.773
C02548=1040.792,-70.739,-76.453,168.988,35.946,156.773
C02549=1040.786,-70.988,-76.442,168.986,35.946,156.773
C02550=1040.780,-71.238,-76.430,168.984,35.945,156.773
C02551=1040.773,-71.487,-76.419,168.981,35.945,156.773
C02552=1040.768,-71.738,-76.407,168.979,35.945,156.773
C02553=1040.761,-71.987,-76.395,168.977,35.944,156.773
C02554=1040.755,-72.237,-76.384,168.974,35.944,156.773
C02555=1040.749,-72.486,-76.372,168.972,35.944,156.773
C02556=1040.743,-72.736,-76.361,168.970,35.944,156.773
C02557=1040.737,-72.986,-76.350,168.967,35.944,156.773
C02558=1040.731,-73.235,-76.338,168.965,35.943,156.772
C02559=1040.725,-73.486,-76.327,168.963,35.943,156.772
C02560=1040.719,-73.734,-76.315,168.960,35.943,156.772
C02561=1040.713,-73.985,-76.303,168.958,35.942,156.772
C02562=1040.707,-74.234,-76.291,168.956,35.942,156.772
C02563=1040.701,-74.484,-76.280,168.953,35.942,156.772
C02564=1040.694,-74.734,-76.270,168.951,35.942,156.772
C02565=1040.688,-74.983,-76.258,168.948,35.941,156.772
C02566=1040.682,-75.233,-76.247,168.946,35.941,156.772
C02567=1040.676,-75.482,-76.236,168.944,35.941,156.772
C02568=1040.669,-75.732,-76.224,168.941,35.941,156.772
C02569=1040.663,-75.982,-76.213,168.939,35.941,156.772
C02570=1040.657,-76.232,-76.202,168.936,35.941,156.772
C02571=1040.651,-76.482,-76.191,168.934,35.941,156.772
C02572=1040.645,-76.731,-76.179,168.932,35.941,156.772
C02573=1040.638,-76.981,-76.168,168.929,35.941,156.772
C02574=1040.633,-77.230,-76.157,168.927,35.941,156.772
C02575=1040.626,-77.480,-76.145,168.924,35.940,156.772
C02576=1040.620,-77.729,-76.134,168.922,35.940,156.772
C02577=1040.614,-77.980,-76.123,168.920,35.940,156.772
C02578=1040.608,-78.229,-76.112,168.917,35.940,156.772
C02579=1040.602,-78.479,-76.100,168.915,35.940,156.772
C02580=1040.596,-78.728,-76.089,168.912,35.940,156.772
C02581=1040.589,-78.978,-76.078,168.910,35.940,156.772
C02582=1040.584,-79.228,-76.067,168.908,35.940,156.772
C02583=1040.577,-79.478,-76.056,168.905,35.940,156.772
C02584=1040.571,-79.727,-76.045,168.903,35.939,156.772
C02585=1040.564,-79.977,-76.034,168.900,35.939,156.772
C02586=1040.559,-80.226,-76.023,168.898,35.939,156.772
C02587=1040.552,-80.477,-76.011,168.896,35.939,156.772
C02588=1040.546,-80.726,-76.001,168.893,35.939,156.772
C02589=1040.539,-80.976,-75.990,168.891,35.939,156.772
C02590=1040.534,-81.225,-75.979,168.888,35.939,156.772
C02591=1040.527,-81.475,-75.968,168.886,35.939,156.772
C02592=1040.521,-81.725,-75.958,168.883,35.939,156.772
C02593=1040.514,-81.975,-75.946,168.881,35.939,156.772
C02594=1040.508,-82.223,-75.935,168.878,35.939,156.772
C02595=1040.502,-82.473,-75.924,168.876,35.939,156.772
C02596=1040.496,-82.723,-75.913,168.874,35.939,156.772
C02597=1040.490,-82.973,-75.902,168.871,35.939,156.772
C02598=1040.483,-83.223,-75.892,168.869,35.939,156.772
C02599=1040.476,-83.507,-75.880,168.866,35.939,156.772
C02600=1040.469,-83.793,-75.867,168.863,35.939,156.772
C02601=1040.461,-84.078,-75.855,168.860,35.939,156.772
C02602=1040.454,-84.362,-75.842,168.858,35.939,156.772
C02603=1040.448,-84.612,-75.831,168.855,35.939,156.772
C02604=1040.442,-84.862,-75.820,168.853,35.939,156.772
C02605=1040.436,-85.111,-75.810,168.850,35.939,156.773
C02606=1040.429,-85.361,-75.799,168.848,35.939,156.773
C02607=1040.424,-85.611,-75.789,168.845,35.939,156.773
C02608=1040.417,-85.861,-75.778,168.843,35.939,156.773
C02609=1040.411,-86.110,-75.767,168.840,35.939,156.773
C02610=1040.405,-86.360,-75.756,168.838,35.939,156.773
C02611=1040.398,-86.610,-75.746,168.835,35.939,156.773
C02612=1040.393,-86.859,-75.735,168.833,35.939,156.773
C02613=1040.387,-87.109,-75.724,168.831,35.939,156.773
C02614=1040.380,-87.359,-75.713,168.828,35.940,156.773
C02615=1040.374,-87.608,-75.702,168.826,35.940,156.773
C02616=1040.368,-87.858,-75.691,168.823,35.940,156.773
C02617=1040.361,-88.108,-75.681,168.821,35.940,156.773
C02618=1040.356,-88.358,-75.671,168.818,35.940,156.773
C02619=1040.350,-88.607,-75.660,168.816,35.939,156.773
C02620=1040.343,-88.857,-75.649,168.813,35.939,156.773
C02621=1040.337,-89.106,-75.638,168.811,35.939,156.773
C02622=1040.331,-89.356,-75.628,168.808,35.940,156.773
C02623=1040.324,-89.606,-75.617,168.806,35.940,156.773
C02624=1040.319,-89.856,-75.607,168.803,35.940,156.773
C02625=1040.313,-90.105,-75.596,168.801,35.940,156.773
C02626=1040.307,-90.355,-75.585,168.798,35.940,156.773
C02627=1040.300,-90.605,-75.575,168.796,35.940,156.773
C02628=1040.294,-90.855,-75.565,168.794,35.940,156.773
C02629=1040.289,-91.104,-75.554,168.791,35.940,156.773
C02630=1040.282,-91.353,-75.543,168.789,35.940,156.773
C02631=1040.276,-91.603,-75.532,168.786,35.940,156.773
C02632=1040.270,-91.854,-75.522,168.784,35.940,156.773
C02633=1040.264,-92.103,-75.512,168.781,35.940,156.773
C02634=1040.258,-92.352,-75.501,168.779,35.940,156.773
C02635=1040.251,-92.602,-75.490,168.776,35.941,156.773
C02636=1040.246,-92.852,-75.480,168.774,35.941,156.773
C02637=1040.239,-93.101,-75.470,168.771,35.941,156.773
C02638=1040.233,-93.351,-75.459,168.769,35.941,156.773
C02639=1040.228,-93.601,-75.449,168.766,35.941,156.773
C02640=1040.221,-93.851,-75.438,168.764,35.941,156.773
C02641=1040.215,-94.100,-75.427,168.761,35.941,156.773
C02642=1040.209,-94.350,-75.418,168.759,35.941,156.773
C02643=1040.203,-94.600,-75.407,168.756,35.941,156.773
C02644=1040.197,-94.849,-75.396,168.754,35.941,156.773
C02645=1040.191,-95.100,-75.386,168.751,35.942,156.774
C02646=1040.185,-95.349,-75.375,168.749,35.942,156.774
C02647=1040.179,-95.598,-75.365,168.746,35.942,156.774
C02648=1040.173,-95.848,-75.355,168.744,35.942,156.774
C02649=1040.167,-96.098,-75.344,168.742,35.942,156.774
C02650=1040.161,-96.348,-75.334,168.740,35.942,156.774
C02651=1040.155,-96.597,-75.323,168.738,35.942,156.774
C02652=1040.148,-96.847,-75.313,168.735,35.942,156.774
C02653=1040.143,-97.097,-75.303,168.733,35.942,156.774
C02654=1040.136,-97.346,-75.292,168.730,35.943,156.774
C02655=1040.131,-97.597,-75.282,168.728,35.943,156.774
C02656=1040.125,-97.846,-75.272,168.725,35.943,156.774
C02657=1040.118,-98.095,-75.262,168.723,35.943,156.774
C02658=1040.113,-98.345,-75.251,168.720,35.943,156.774
C02659=1040.106,-98.595,-75.241,168.718,35.943,156.774
C02660=1040.099,-98.845,-75.231,168.715,35.944,156.774
C02661=1040.094,-99.095,-75.221,168.712,35.944,156.774
C02662=1040.088,-99.345,-75.211,168.710,35.944,156.774
C02663=1040.081,-99.585,-75.202,168.708,35.944,156.774
C02664=1040.076,-99.826,-75.191,168.705,35.945,156.774
C02665=1040.069,-100.067,-75.182,168.703,35.945,156.774
C02666=1040.064,-100.308,-75.172,168.700,35.945,156.774
C02667=1040.058,-100.548,-75.162,168.698,35.946,156.775
C02668=1040.053,-100.790,-75.153,168.695,35.945,156.775
C02669=1040.046,-101.030,-75.143,168.693,35.946,156.775
C02670=1040.041,-101.271,-75.133,168.690,35.946,156.775
C02671=1040.034,-101.521,-75.123,168.688,35.947,156.775
C02672=1040.028,-101.770,-75.114,168.685,35.947,156.775
C02673=1040.023,-102.020,-75.103,168.683,35.947,156.775
C02674=1040.016,-102.270,-75.093,168.680,35.947,156.775
C02675=1040.010,-102.520,-75.083,168.678,35.947,156.775
C02676=1040.003,-102.769,-75.073,168.675,35.948,156.775
C02677=1039.998,-103.019,-75.063,168.673,35.948,156.775
C02678=1039.991,-103.269,-75.053,168.670,35.948,156.775
C02679=1039.985,-103.518,-75.043,168.668,35.948,156.775
C02680=1039.979,-103.768,-75.034,168.665,35.949,156.775
C02681=1039.973,-104.018,-75.023,168.663,35.949,156.775
C02682=1039.967,-104.267,-75.013,168.660,35.950,156.775
C02683=1039.961,-104.517,-75.004,168.658,35.950,156.775
C02684=1039.955,-104.767,-74.994,168.656,35.950,156.776
C02685=1039.949,-105.017,-74.984,168.653,35.950,156.776
C02686=1039.943,-105.266,-74.974,168.651,35.951,156.776
C02687=1039.937,-105.516,-74.964,168.648,35.951,156.776
C02688=1039.930,-105.766,-74.954,168.646,35.951,156.776
C02689=1039.925,-106.016,-74.944,168.643,35.952,156.776
C02690=1039.919,-106.266,-74.935,168.641,35.952,156.776
C02691=1039.912,-106.515,-74.924,168.638,35.952,156.776
C02692=1039.906,-106.765,-74.915,168.636,35.952,156.776
C02693=1039.900,-107.015,-74.905,168.633,35.953,156.776
C02694=1039.894,-107.265,-74.895,168.631,35.953,156.776
C02695=1039.888,-107.515,-74.886,168.628,35.954,156.776
C02696=1039.882,-107.764,-74.876,168.625,35.954,156.776
C02697=1039.876,-108.014,-74.866,168.623,35.954,156.776
C02698=1039.869,-108.263,-74.856,168.620,35.955,156.777
C02699=1039.863,-108.513,-74.847,168.618,35.955,156.777
C02700=1039.857,-108.763,-74.837,168.615,35.955,156.777
C02701=1039.852,-109.012,-74.828,168.613,35.956,156.777
C02702=1039.845,-109.262,-74.818,168.610,35.957,156.777
C02703=1039.840,-109.512,-74.808,168.607,35.957,156.777
C02704=1039.834,-109.762,-74.798,168.605,35.957,156.777
C02705=1039.828,-110.012,-74.789,168.602,35.958,156.777
C02706=1039.821,-110.261,-74.779,168.600,35.958,156.777
C02707=1039.814,-110.566,-74.767,168.597,35.958,156.777
C02708=1039.806,-110.871,-74.756,168.594,35.959,156.777
C02709=1039.799,-111.176,-74.744,168.591,35.960,156.778
C02710=1039.792,-111.481,-74.732,168.588,35.960,156.778
C02711=1039.785,-111.730,-74.722,168.586,35.960,156.778
C02712=1039.779,-111.980,-74.713,168.583,35.961,156.778
C02713=1039.773,-112.231,-74.704,168.580,35.961,156.778
C02714=1039.767,-112.480,-74.694,168.578,35.962,156.778
C02715=1039.761,-112.730,-74.685,168.575,35.962,156.778
C02716=1039.755,-112.980,-74.675,168.573,35.963,156.778
C02717=1039.749,-113.229,-74.666,168.570,35.963,156.778
C02718=1039.743,-113.479,-74.657,168.568,35.963,156.778
C02719=1039.737,-113.729,-74.647,168.565,35.964,156.778
C02720=1039.731,-113.978,-74.637,168.562,35.964,156.779
C02721=1039.725,-114.228,-74.628,168.560,35.965,156.779
C02722=1039.718,-114.478,-74.618,168.557,35.965,156.779
///RCONF 1,0,0,0,1,0,0,0,0,0,0,0,0,0,0,0,0,0,0,0,0,0,0,0
C02723=1039.712,-114.728,-74.609,168.555,35.966,156.779
C02724=1039.707,-114.977,-74.600,168.552,35.966,156.779
C02725=1039.701,-115.227,-74.590,168.549,35.967,156.779
C02726=1039.695,-115.477,-74.581,168.547,35.967,156.779
C02727=1039.688,-115.763,-74.570,168.544,35.968,156.779
C02728=1039.680,-116.049,-74.559,168.542,35.969,156.779
C02729=1039.673,-116.336,-74.548,168.539,35.969,156.780
C02730=1039.667,-116.623,-74.538,168.536,35.970,156.780
C02731=1039.660,-116.871,-74.529,168.533,35.970,156.780
C02732=1039.654,-117.121,-74.519,168.531,35.971,156.780
C02733=1039.648,-117.372,-74.511,168.528,35.971,156.780
C02734=1039.642,-117.621,-74.501,168.526,35.972,156.780
C02735=1039.637,-117.871,-74.492,168.523,35.972,156.780
C02736=1039.631,-118.120,-74.482,168.520,35.973,156.780
C02737=1039.625,-118.371,-74.473,168.518,35.974,156.780
C02738=1039.618,-118.621,-74.464,168.515,35.974,156.781
C02739=1039.612,-118.870,-74.454,168.513,35.975,156.781
C02740=1039.606,-119.119,-74.446,168.510,35.975,156.781
C02741=1039.600,-119.370,-74.437,168.507,35.975,156.781
C02742=1039.594,-119.619,-74.427,168.505,35.976,156.781
C02743=1039.588,-119.869,-74.418,168.502,35.977,156.781
C02744=1039.583,-120.119,-74.409,168.500,35.977,156.781
C02745=1039.576,-120.369,-74.400,168.497,35.978,156.781
C02746=1039.569,-120.618,-74.391,168.495,35.979,156.781
C02747=1039.564,-120.868,-74.382,168.493,35.979,156.781
C02748=1039.558,-121.118,-74.373,168.490,35.980,156.782
C02749=1039.552,-121.367,-74.363,168.487,35.980,156.782
C02750=1039.546,-121.618,-74.354,168.485,35.981,156.782
C02751=1039.540,-121.867,-74.345,168.482,35.982,156.782
C02752=1039.533,-122.116,-74.336,168.480,35.982,156.782
C02753=1039.528,-122.367,-74.327,168.477,35.983,156.782
C02754=1039.522,-122.616,-74.318,168.474,35.983,156.782
C02755=1039.516,-122.866,-74.309,168.472,35.984,156.782
C02756=1039.510,-123.116,-74.299,168.469,35.985,156.783
C02757=1039.504,-123.365,-74.291,168.467,35.985,156.783
C02758=1039.498,-123.615,-74.282,168.464,35.986,156.783
C02759=1039.492,-123.865,-74.272,168.461,35.987,156.783
C02760=1039.486,-124.115,-74.264,168.459,35.987,156.783
C02761=1039.479,-124.364,-74.255,168.456,35.988,156.783
C02762=1039.474,-124.615,-74.246,168.454,35.988,156.783
C02763=1039.468,-124.864,-74.237,168.452,35.989,156.783
C02764=1039.461,-125.114,-74.229,168.449,35.990,156.784
C02765=1039.455,-125.364,-74.219,168.447,35.990,156.784
C02766=1039.450,-125.614,-74.211,168.444,35.991,156.784
C02767=1039.443,-125.863,-74.202,168.441,35.992,156.784
C02768=1039.437,-126.113,-74.193,168.439,35.993,156.784
C02769=1039.432,-126.363,-74.184,168.436,35.993,156.784
C02770=1039.425,-126.613,-74.175,168.433,35.994,156.784
C02771=1039.419,-126.862,-74.166,168.431,35.995,156.784
C02772=1039.414,-127.112,-74.157,168.428,35.995,156.785
C02773=1039.407,-127.362,-74.149,168.425,35.996,156.785
C02774=1039.401,-127.611,-74.140,168.423,35.997,156.785
C02775=1039.396,-127.862,-74.131,168.420,35.998,156.785
C02776=1039.390,-128.111,-74.122,168.418,35.998,156.785
C02777=1039.386,-128.361,-74.111,168.415,35.998,156.785
C02778=1039.382,-128.610,-74.101,168.413,35.997,156.785
C02779=1039.379,-128.861,-74.089,168.411,35.996,156.785
C02780=1039.377,-129.110,-74.078,168.409,35.994,156.785
C02781=1039.376,-129.360,-74.065,168.407,35.992,156.784
C02782=1039.376,-129.610,-74.053,168.406,35.990,156.784
C02783=1039.376,-129.860,-74.039,168.404,35.987,156.783
C02784=1039.378,-130.110,-74.024,168.402,35.983,156.783
C02785=1039.379,-130.361,-74.010,168.401,35.980,156.782
C02786=1039.382,-130.610,-73.995,168.400,35.975,156.781
C02787=1039.385,-130.861,-73.979,168.398,35.971,156.781
C02788=1039.390,-131.111,-73.962,168.397,35.965,156.780
C02789=1039.395,-131.361,-73.945,168.396,35.959,156.779
C02790=1039.401,-131.611,-73.927,168.395,35.954,156.778
C02791=1039.057,-131.635,-74.190,168.347,36.153,156.812
C02792=1039.051,-131.385,-74.208,168.348,36.160,156.813
C02793=1039.046,-131.135,-74.225,168.349,36.165,156.814
C02794=1039.042,-130.885,-74.242,168.351,36.170,156.814
C02795=1039.038,-130.634,-74.259,168.352,36.176,156.815
C02796=1039.035,-130.384,-74.274,168.354,36.180,156.816
C02797=1039.033,-130.134,-74.288,168.355,36.183,156.817
C02798=1039.032,-129.885,-74.302,168.356,36.187,156.817
C02799=1039.032,-129.635,-74.316,168.358,36.189,156.818
C02800=1039.032,-129.384,-74.329,168.360,36.192,156.818
C02801=1039.033,-129.135,-74.341,168.362,36.194,156.818
C02802=1039.035,-128.884,-74.354,168.364,36.196,156.819
C02803=1039.038,-128.635,-74.364,168.366,36.197,156.819
C02804=1039.041,-128.385,-74.375,168.368,36.197,156.819
C02805=1039.046,-128.135,-74.385,168.370,36.198,156.819
C02806=1039.052,-127.885,-74.395,168.373,36.197,156.819
C02807=1039.057,-127.636,-74.404,168.375,36.197,156.819
C02808=1039.063,-127.387,-74.412,168.378,36.196,156.819
C02809=1039.069,-127.136,-74.421,168.381,36.196,156.819
C02810=1039.075,-126.886,-74.430,168.383,36.195,156.819
C02811=1039.081,-126.637,-74.439,168.386,36.194,156.818
C02812=1039.087,-126.387,-74.447,168.389,36.193,156.818
C02813=1039.093,-126.138,-74.457,168.391,36.192,156.818
C02814=1039.099,-125.888,-74.465,168.394,36.192,156.818
C02815=1039.105,-125.638,-74.474,168.397,36.191,156.818
C02816=1039.111,-125.388,-74.483,168.399,36.190,156.818
C02817=1039.118,-125.139,-74.492,168.402,36.189,156.817
C02818=1039.123,-124.888,-74.501,168.404,36.188,156.817
C02819=1039.129,-124.639,-74.510,168.406,36.188,156.817
C02820=1039.136,-124.389,-74.518,168.409,36.187,156.817
C02821=1039.142,-124.139,-74.528,168.412,36.187,156.817
C02822=1039.147,-123.889,-74.536,168.414,36.186,156.817
C02823=1039.153,-123.640,-74.546,168.417,36.185,156.817
C02824=1039.160,-123.390,-74.554,168.419,36.185,156.817
C02825=1039.165,-123.141,-74.563,168.422,36.184,156.817
C02826=1039.171,-122.890,-74.572,168.425,36.183,156.816
C02827=1039.177,-122.640,-74.582,168.427,36.183,156.816
C02828=1039.183,-122.391,-74.591,168.430,36.182,156.816
C02829=1039.190,-122.141,-74.599,168.433,36.181,156.816
C02830=1039.196,-121.891,-74.609,168.435,36.181,156.816
C02831=1039.201,-121.642,-74.617,168.438,36.180,156.816
C02832=1039.207,-121.392,-74.627,168.440,36.180,156.816
C02833=1039.213,-121.142,-74.636,168.443,36.179,156.816
C02834=1039.220,-120.892,-74.645,168.445,36.178,156.815
C02835=1039.226,-120.643,-74.654,168.447,36.178,156.815
C02836=1039.232,-120.393,-74.663,168.450,36.177,156.815
C02837=1039.238,-120.143,-74.672,168.453,36.176,156.815
C02838=1039.243,-119.893,-74.681,168.455,36.176,156.815
C02839=1039.249,-119.644,-74.691,168.458,36.175,156.815
C02840=1039.256,-119.394,-74.699,168.460,36.175,156.815
C02841=1039.262,-119.144,-74.709,168.463,36.174,156.815
C02842=1039.268,-118.895,-74.718,168.466,36.173,156.815
C02843=1039.274,-118.645,-74.728,168.468,36.173,156.814
C02844=1039.280,-118.394,-74.736,168.471,36.172,156.814
C02845=1039.286,-118.145,-74.746,168.474,36.171,156.814
C02846=1039.291,-117.896,-74.755,168.476,36.171,156.814
C02847=1039.298,-117.646,-74.764,168.479,36.170,156.814
C02848=1039.304,-117.396,-74.773,168.481,36.169,156.814
C02849=1039.310,-117.146,-74.783,168.484,36.169,156.814
C02850=1039.317,-116.896,-74.792,168.486,36.168,156.814
C02851=1039.322,-116.647,-74.801,168.488,36.168,156.814
C02852=1039.329,-116.360,-74.812,168.491,36.167,156.813
C02853=1039.336,-116.074,-74.823,168.494,36.166,156.813
C02854=1039.343,-115.787,-74.833,168.497,36.166,156.813
C02855=1039.350,-115.501,-74.844,168.500,36.165,156.813
C02856=1039.356,-115.251,-74.854,168.503,36.165,156.813
C02857=1039.362,-115.002,-74.862,168.505,36.164,156.813
C02858=1039.368,-114.752,-74.872,168.508,36.164,156.813
C02859=1039.375,-114.503,-74.882,168.511,36.163,156.813
C02860=1039.381,-114.253,-74.891,168.513,36.163,156.813
C02861=1039.387,-114.002,-74.900,168.516,36.162,156.812
C02862=1039.393,-113.753,-74.910,168.519,36.162,156.812
C02863=1039.399,-113.503,-74.919,168.521,36.161,156.812
C02864=1039.405,-113.254,-74.928,168.524,36.161,156.812
C02865=1039.411,-113.004,-74.938,168.526,36.160,156.812
C02866=1039.416,-112.754,-74.948,168.529,36.159,156.812
///RCONF 1,0,0,0,0,0,0,0,0,0,0,0,0,0,0,0,0,0,0,0,0,0,0,0
C02867=1039.422,-112.504,-74.958,168.531,36.159,156.812
C02868=1039.428,-112.254,-74.967,168.533,36.159,156.812
C02869=1039.435,-112.004,-74.977,168.536,36.158,156.812
C02870=1039.441,-111.755,-74.986,168.538,36.158,156.812
C02871=1039.446,-111.506,-74.996,168.541,36.158,156.812
C02872=1039.453,-111.256,-75.005,168.543,36.157,156.811
C02873=1039.459,-111.006,-75.015,168.546,36.156,156.811
C02874=1039.465,-110.756,-75.024,168.549,36.156,156.811
C02875=1039.471,-110.506,-75.034,168.551,36.156,156.811
C02876=1039.477,-110.257,-75.043,168.554,36.155,156.811
C02877=1039.483,-110.007,-75.053,168.556,36.154,156.811
C02878=1039.490,-109.757,-75.063,168.559,36.154,156.811
C02879=1039.496,-109.507,-75.072,168.562,36.154,156.811
C02880=1039.502,-109.257,-75.082,168.564,36.153,156.811
C02881=1039.508,-109.008,-75.091,168.567,36.153,156.811
C02882=1039.514,-108.757,-75.101,168.569,36.153,156.811
C02883=1039.520,-108.508,-75.111,168.572,36.152,156.811
C02884=1039.526,-108.259,-75.121,168.574,36.151,156.810
C02885=1039.532,-108.009,-75.130,168.577,36.151,156.810
C02886=1039.538,-107.760,-75.140,168.580,36.151,156.810
C02887=1039.544,-107.510,-75.150,168.582,36.150,156.810
C02888=1039.550,-107.260,-75.159,168.585,36.150,156.810
C02889=1039.556,-107.010,-75.169,168.587,36.149,156.810
C02890=1039.562,-106.760,-75.179,168.589,36.149,156.810
C02891=1039.568,-106.511,-75.189,168.591,36.149,156.810
C02892=1039.575,-106.261,-75.199,168.594,36.148,156.810
C02893=1039.581,-106.011,-75.208,168.597,36.148,156.810
C02894=1039.587,-105.762,-75.218,168.599,36.148,156.810
C02895=1039.592,-105.511,-75.228,168.602,36.147,156.810
C02896=1039.599,-105.262,-75.238,168.604,36.147,156.810
C02897=1039.605,-105.012,-75.248,168.607,36.146,156.809
C02898=1039.611,-104.763,-75.257,168.609,36.146,156.809
C02899=1039.617,-104.513,-75.268,168.612,36.146,156.809
C02900=1039.623,-104.263,-75.278,168.615,36.146,156.809
C02901=1039.629,-104.014,-75.287,168.617,36.145,156.809
C02902=1039.635,-103.764,-75.297,168.620,36.145,156.809
C02903=1039.641,-103.514,-75.307,168.622,36.145,156.809
C02904=1039.647,-103.264,-75.317,168.625,36.144,156.809
C02905=1039.653,-103.015,-75.327,168.627,36.144,156.809
C02906=1039.660,-102.765,-75.337,168.630,36.143,156.809
C02907=1039.665,-102.515,-75.347,168.632,36.143,156.809
C02908=1039.672,-102.265,-75.357,168.635,36.143,156.809
C02909=1039.678,-102.015,-75.367,168.637,36.143,156.809
C02910=1039.684,-101.766,-75.378,168.640,36.142,156.809
C02911=1039.690,-101.516,-75.387,168.643,36.142,156.809
C02912=1039.696,-101.266,-75.397,168.645,36.142,156.808
C02913=1039.702,-101.017,-75.408,168.648,36.142,156.808
C02914=1039.708,-100.767,-75.417,168.650,36.141,156.808
C02915=1039.714,-100.517,-75.427,168.653,36.141,156.808
C02916=1039.722,-100.230,-75.439,168.656,36.140,156.808
C02917=1039.729,-99.943,-75.451,168.658,36.140,156.808
C02918=1039.736,-99.655,-75.462,168.660,36.140,156.808
C02919=1039.743,-99.368,-75.475,168.663,36.140,156.808
C02920=1039.749,-99.118,-75.484,168.666,36.139,156.808
C02921=1039.755,-98.869,-75.494,168.668,36.139,156.808
C02922=1039.762,-98.619,-75.504,168.671,36.139,156.808
C02923=1039.767,-98.369,-75.514,168.674,36.139,156.808
C02924=1039.774,-98.120,-75.524,168.676,36.138,156.808
C02925=1039.780,-97.870,-75.534,168.679,36.138,156.808
C02926=1039.786,-97.620,-75.545,168.681,36.137,156.808
C02927=1039.792,-97.370,-75.555,168.684,36.137,156.808
C02928=1039.798,-97.121,-75.566,168.686,36.137,156.808
C02929=1039.804,-96.871,-75.575,168.689,36.137,156.807
C02930=1039.810,-96.622,-75.586,168.691,36.137,156.807
C02931=1039.816,-96.372,-75.596,168.694,36.137,156.807
C02932=1039.822,-96.122,-75.607,168.696,36.137,156.807
C02933=1039.828,-95.873,-75.617,168.699,36.136,156.807
C02934=1039.834,-95.622,-75.627,168.701,36.136,156.807
C02935=1039.840,-95.373,-75.638,168.704,36.136,156.807
C02936=1039.847,-95.124,-75.649,168.706,36.136,156.807
C02937=1039.852,-94.874,-75.659,168.709,36.136,156.807
C02938=1039.858,-94.624,-75.669,168.711,36.136,156.807
C02939=1039.864,-94.374,-75.679,168.714,36.136,156.807
C02940=1039.870,-94.124,-75.690,168.716,36.136,156.807
C02941=1039.877,-93.875,-75.701,168.719,36.135,156.807
C02942=1039.882,-93.625,-75.711,168.721,36.135,156.807
C02943=1039.889,-93.376,-75.721,168.724,36.135,156.807
C02944=1039.899,-92.954,-75.739,168.728,36.135,156.807
C02945=1039.909,-92.532,-75.758,168.732,36.135,156.807
C02946=1039.919,-92.110,-75.775,168.736,36.135,156.807
C02947=1039.930,-91.688,-75.793,168.740,36.134,156.807
C02948=1039.936,-91.439,-75.803,168.743,36.134,156.807
C02949=1039.942,-91.189,-75.813,168.745,36.134,156.807
C02950=1039.947,-90.939,-75.824,168.748,36.134,156.807
C02951=1039.955,-90.689,-75.835,168.750,36.134,156.807
C02952=1039.960,-90.440,-75.846,168.753,36.133,156.807
C02953=1039.966,-90.190,-75.856,168.755,36.134,156.807
C02954=1039.972,-89.941,-75.866,168.758,36.134,156.807
C02955=1039.979,-89.690,-75.877,168.760,36.134,156.807
C02956=1039.985,-89.441,-75.888,168.763,36.134,156.807
C02957=1039.991,-89.192,-75.898,168.765,36.133,156.806
C02958=1039.997,-88.942,-75.910,168.768,36.133,156.806
C02959=1040.003,-88.692,-75.919,168.770,36.133,156.806
C02960=1040.009,-88.442,-75.930,168.773,36.133,156.806
C02961=1040.015,-88.193,-75.941,168.775,36.133,156.806
C02962=1040.022,-87.943,-75.952,168.778,36.133,156.806
C02963=1040.028,-87.693,-75.962,168.779,36.132,156.806
C02964=1040.034,-87.444,-75.973,168.782,36.132,156.806
C02965=1040.040,-87.194,-75.984,168.784,36.132,156.806
C02966=1040.046,-86.944,-75.994,168.787,36.133,156.806
C02967=1040.052,-86.695,-76.004,168.789,36.133,156.806
C02968=1040.059,-86.445,-76.016,168.792,36.133,156.806
C02969=1040.064,-86.195,-76.027,168.794,36.132,156.806
C02970=1040.071,-85.945,-76.037,168.796,36.132,156.806
C02971=1040.077,-85.696,-76.048,168.799,36.132,156.806
C02972=1040.083,-85.446,-76.059,168.801,36.132,156.806
C02973=1040.090,-85.196,-76.070,168.804,36.132,156.806
C02974=1040.096,-84.947,-76.080,168.806,36.132,156.806
C02975=1040.101,-84.697,-76.091,168.809,36.132,156.806
C02976=1040.111,-84.334,-76.107,168.812,36.131,156.806
C02977=1040.120,-83.972,-76.123,168.816,36.132,156.806
C02978=1040.129,-83.609,-76.138,168.820,36.132,156.806
C02979=1040.139,-83.247,-76.154,168.823,36.132,156.806
C02980=1040.144,-82.997,-76.165,168.826,36.132,156.806
C02981=1040.150,-82.748,-76.176,168.828,36.132,156.806
C02982=1040.157,-82.498,-76.187,168.831,36.132,156.806
C02983=1040.163,-82.248,-76.198,168.833,36.131,156.806
C02984=1040.169,-81.998,-76.209,168.835,36.131,156.806
C02985=1040.176,-81.749,-76.219,168.838,36.131,156.806
C02986=1040.182,-81.499,-76.230,168.840,36.131,156.806
C02987=1040.188,-81.249,-76.241,168.843,36.131,156.806
C02988=1040.195,-80.999,-76.252,168.845,36.131,156.806
C02989=1040.201,-80.750,-76.263,168.848,36.131,156.806
C02990=1040.207,-80.500,-76.275,168.850,36.131,156.806
C02991=1040.214,-80.251,-76.285,168.853,36.131,156.806
C02992=1040.220,-80.001,-76.296,168.855,36.131,156.806
C02993=1040.226,-79.751,-76.307,168.858,36.131,156.806
C02994=1040.232,-79.501,-76.318,168.860,36.131,156.806
C02995=1040.238,-79.252,-76.329,168.862,36.131,156.806
C02996=1040.245,-79.002,-76.341,168.865,36.131,156.806
C02997=1040.250,-78.753,-76.352,168.867,36.131,156.806
C02998=1040.257,-78.502,-76.363,168.870,36.131,156.806
C02999=1040.262,-78.253,-76.374,168.872,36.131,156.806
C03000=1040.269,-78.003,-76.385,168.874,36.131,156.806
C03001=1040.276,-77.754,-76.396,168.877,36.131,156.806
C03002=1040.282,-77.504,-76.408,168.879,36.131,156.806
C03003=1040.288,-77.254,-76.418,168.882,36.132,156.806
C03004=1040.294,-77.004,-76.430,168.884,36.132,156.806
C03005=1040.300,-76.755,-76.441,168.887,36.132,156.806
C03006=1040.306,-76.505,-76.453,168.889,36.132,156.806
C03007=1040.312,-76.256,-76.463,168.891,36.132,156.806
C03008=1040.319,-76.006,-76.475,168.894,36.132,156.806
C03009=1040.324,-75.757,-76.486,168.896,36.132,156.806
C03010=1040.331,-75.506,-76.498,168.899,36.132,156.806
C03011=1040.337,-75.258,-76.509,168.901,36.132,156.806
C03012=1040.343,-75.007,-76.520,168.903,36.133,156.806
C03013=1040.349,-74.758,-76.531,168.906,36.133,156.806
C03014=1040.356,-74.508,-76.543,168.908,36.133,156.806
C03015=1040.362,-74.258,-76.554,168.911,36.133,156.806
C03016=1040.368,-74.009,-76.565,168.913,36.133,156.806
C03017=1040.374,-73.759,-76.577,168.915,36.133,156.806
C03018=1040.380,-73.510,-76.588,168.918,36.134,156.806
C03019=1040.386,-73.259,-76.599,168.920,36.134,156.806
C03020=1040.392,-73.010,-76.612,168.922,36.134,156.806
C03021=1040.398,-72.760,-76.623,168.925,36.135,156.806
C03022=1040.405,-72.510,-76.635,168.927,36.135,156.806
C03023=1040.410,-72.261,-76.646,168.929,36.135,156.806
C03024=1040.417,-72.011,-76.658,168.932,36.135,156.806
C03025=1040.422,-71.762,-76.669,168.934,36.135,156.806
C03026=1040.429,-71.512,-76.681,168.937,36.135,156.806
C03027=1040.434,-71.263,-76.692,168.939,36.136,156.806
C03028=1040.441,-71.013,-76.704,168.941,36.136,156.806
C03029=1040.447,-70.762,-76.716,168.944,36.136,156.806
C03030=1040.453,-70.514,-76.727,168.946,36.137,156.806
C03031=1040.459,-70.263,-76.739,168.948,36.137,156.806
C03032=1040.465,-70.015,-76.750,168.951,36.137,156.806
C03033=1040.471,-69.765,-76.763,168.954,36.137,156.806
C03034=1040.477,-69.514,-76.774,168.956,36.137,156.806
C03035=1040.483,-69.266,-76.786,168.959,36.137,156.806
C03036=1040.490,-69.015,-76.797,168.961,36.138,156.807
C03037=1040.495,-68.766,-76.809,168.963,36.138,156.807
C03038=1040.501,-68.516,-76.820,168.966,36.139,156.807
C03039=1040.508,-68.266,-76.832,168.968,36.139,156.807
C03040=1040.515,-67.984,-76.845,168.971,36.139,156.807
C03041=1040.522,-67.701,-76.858,168.973,36.140,156.807
C03042=1040.529,-67.418,-76.872,168.976,36.140,156.807
C03043=1040.536,-67.136,-76.885,168.979,36.140,156.807
C03044=1040.543,-66.886,-76.897,168.981,36.140,156.807
C03045=1040.548,-66.636,-76.909,168.983,36.140,156.807
C03046=1040.554,-66.387,-76.921,168.986,36.141,156.807
C03047=1040.561,-66.137,-76.933,168.988,36.141,156.807
C03048=1040.566,-65.887,-76.944,168.990,36.141,156.807
C03049=1040.573,-65.638,-76.956,168.993,36.142,156.807
C03050=1040.579,-65.388,-76.968,168.995,36.142,156.807
C03051=1040.585,-65.139,-76.979,168.997,36.142,156.807
C03052=1040.591,-64.889,-76.991,169.000,36.142,156.807
C03053=1040.597,-64.639,-77.003,169.002,36.142,156.807
C03054=1040.604,-64.390,-77.015,169.004,36.143,156.807
C03055=1040.609,-64.140,-77.027,169.007,36.143,156.807
C03056=1040.616,-63.890,-77.039,169.009,36.144,156.807
C03057=1040.622,-63.641,-77.051,169.011,36.144,156.807
C03058=1040.629,-63.391,-77.063,169.014,36.144,156.807
C03059=1040.634,-63.141,-77.074,169.016,36.144,156.807
C03060=1040.641,-62.892,-77.086,169.018,36.144,156.807
C03061=1040.647,-62.642,-77.098,169.021,36.145,156.808
C03062=1040.653,-62.392,-77.111,169.023,36.145,156.808
C03063=1040.659,-62.143,-77.122,169.025,36.145,156.808
C03064=1040.666,-61.893,-77.133,169.028,36.146,156.808
C03065=1040.672,-61.643,-77.146,169.030,36.146,156.808
C03066=1040.678,-61.394,-77.158,169.032,36.147,156.808
C03067=1040.685,-61.144,-77.170,169.035,36.147,156.808
C03068=1040.691,-60.895,-77.182,169.037,36.147,156.808
C03069=1040.697,-60.646,-77.194,169.039,36.147,156.808
C03070=1040.703,-60.395,-77.205,169.042,36.147,156.808
C03071=1040.710,-60.146,-77.217,169.044,36.148,156.808
C03072=1040.716,-59.896,-77.230,169.046,36.148,156.808
C03073=1040.722,-59.646,-77.242,169.049,36.149,156.808
C03074=1040.728,-59.397,-77.253,169.051,36.149,156.808
C03075=1040.734,-59.148,-77.266,169.053,36.149,156.808
C03076=1040.741,-58.898,-77.278,169.055,36.149,156.808
C03077=1040.748,-58.648,-77.290,169.058,36.150,156.808
C03078=1040.753,-58.399,-77.302,169.060,36.150,156.808
C03079=1040.760,-58.149,-77.314,169.062,36.150,156.808
C03080=1040.767,-57.899,-77.326,169.066,36.151,156.808
C03081=1040.773,-57.649,-77.339,169.068,36.151,156.808
C03082=1040.778,-57.400,-77.350,169.070,36.151,156.808
C03083=1040.785,-57.150,-77.362,169.073,36.151,156.808
C03084=1040.791,-56.901,-77.374,169.075,36.152,156.809
C03085=1040.798,-56.651,-77.386,169.077,36.152,156.809
C03086=1040.804,-56.401,-77.399,169.080,36.153,156.809
C03087=1040.810,-56.152,-77.411,169.082,36.153,156.809
C03088=1040.817,-55.902,-77.423,169.084,36.153,156.809
C03089=1040.823,-55.652,-77.435,169.086,36.154,156.809
C03090=1040.830,-55.403,-77.448,169.089,36.154,156.809
C03091=1040.836,-55.154,-77.460,169.091,36.154,156.809
C03092=1040.842,-54.904,-77.472,169.093,36.154,156.809
C03093=1040.849,-54.654,-77.484,169.096,36.155,156.809
C03094=1040.856,-54.405,-77.496,169.098,36.155,156.809
C03095=1040.861,-54.155,-77.509,169.100,36.156,156.809
C03096=1040.868,-53.906,-77.521,169.103,36.156,156.809
C03097=1040.873,-53.656,-77.533,169.105,36.156,156.809
C03098=1040.880,-53.406,-77.545,169.107,36.156,156.809
C03099=1040.887,-53.157,-77.557,169.109,36.157,156.809
C03100=1040.893,-52.907,-77.570,169.112,36.157,156.809
C03101=1040.899,-52.657,-77.582,169.114,36.158,156.809
C03102=1040.906,-52.408,-77.594,169.116,36.158,156.809
C03103=1040.912,-52.158,-77.607,169.119,36.158,156.810
C03104=1040.919,-51.876,-77.620,169.121,36.158,156.810
C03105=1040.927,-51.595,-77.634,169.124,36.159,156.810
C03106=1040.934,-51.313,-77.648,169.126,36.159,156.810
C03107=1040.942,-51.032,-77.662,169.129,36.160,156.810
C03108=1040.948,-50.782,-77.674,169.131,36.160,156.810
C03109=1040.954,-50.532,-77.687,169.133,36.160,156.810
C03110=1040.960,-50.282,-77.700,169.136,36.161,156.810
C03111=1040.967,-50.034,-77.712,169.138,36.161,156.810
C03112=1040.973,-49.784,-77.725,169.140,36.162,156.810
C03113=1040.979,-49.534,-77.737,169.142,36.162,156.810
C03114=1040.986,-49.285,-77.750,169.146,36.163,156.810
C03115=1040.992,-49.035,-77.763,169.148,36.163,156.810
C03116=1040.998,-48.785,-77.775,169.150,36.164,156.810
C03117=1041.004,-48.535,-77.788,169.152,36.164,156.810
C03118=1041.011,-48.286,-77.800,169.154,36.165,156.811
C03119=1041.016,-48.036,-77.813,169.157,36.165,156.811
C03120=1041.022,-47.786,-77.825,169.159,36.166,156.811
C03121=1041.029,-47.537,-77.839,169.161,36.166,156.811
C03122=1041.035,-47.288,-77.851,169.163,36.167,156.811
C03123=1041.041,-47.038,-77.864,169.166,36.167,156.811
C03124=1041.047,-46.788,-77.876,169.168,36.168,156.811
C03125=1041.053,-46.539,-77.889,169.170,36.168,156.811
C03126=1041.060,-46.290,-77.902,169.172,36.169,156.811
C03127=1041.066,-46.040,-77.914,169.174,36.169,156.811
C03128=1041.072,-45.790,-77.928,169.177,36.170,156.811
C03129=1041.078,-45.541,-77.940,169.179,36.170,156.811
C03130=1041.085,-45.291,-77.952,169.181,36.171,156.812
C03131=1041.091,-45.042,-77.965,169.183,36.171,156.812
C03132=1041.097,-44.792,-77.978,169.185,36.172,156.812
C03133=1041.103,-44.543,-77.991,169.188,36.172,156.812
C03134=1041.109,-44.293,-78.004,169.190,36.173,156.812
C03135=1041.117,-44.043,-78.017,169.192,36.173,156.812
C03136=1041.123,-43.793,-78.029,169.194,36.174,156.812
C03137=1041.129,-43.544,-78.043,169.197,36.174,156.812
C03138=1041.135,-43.294,-78.055,169.200,36.175,156.812
C03139=1041.142,-43.045,-78.068,169.202,36.175,156.812
C03140=1041.148,-42.795,-78.080,169.204,36.176,156.812
C03141=1041.154,-42.546,-78.094,169.206,36.176,156.812
C03142=1041.160,-42.296,-78.106,169.209,36.177,156.813
C03143=1041.167,-42.046,-78.120,169.211,36.178,156.813
C03144=1041.173,-41.797,-78.132,169.213,36.178,156.813
C03145=1041.179,-41.547,-78.145,169.215,36.178,156.813
C03146=1041.185,-41.297,-78.158,169.217,36.179,156.813
C03147=1041.191,-41.048,-78.171,169.219,36.180,156.813
C03148=1041.198,-40.799,-78.184,169.222,36.180,156.813
C03149=1041.204,-40.549,-78.196,169.224,36.180,156.813
C03150=1041.211,-40.299,-78.210,169.226,36.181,156.813
C03151=1041.217,-40.049,-78.222,169.228,36.182,156.813
C03152=1041.223,-39.800,-78.236,169.230,36.182,156.813
C03153=1041.229,-39.551,-78.249,169.233,36.182,156.813
C03154=1041.236,-39.301,-78.261,169.235,36.183,156.813
C03155=1041.243,-39.051,-78.274,169.237,36.184,156.814
C03156=1041.249,-38.801,-78.287,169.239,36.184,156.814
C03157=1041.255,-38.552,-78.300,169.241,36.185,156.814
C03158=1041.261,-38.303,-78.313,169.245,36.186,156.814
C03159=1041.267,-38.053,-78.326,169.247,36.186,156.814
C03160=1041.274,-37.803,-78.340,169.249,36.187,156.814
C03161=1041.280,-37.554,-78.353,169.251,36.188,156.814
C03162=1041.286,-37.305,-78.366,169.253,36.188,156.814
C03163=1041.292,-37.055,-78.379,169.255,36.188,156.814
C03164=1041.299,-36.805,-78.392,169.257,36.189,156.814
C03165=1041.305,-36.555,-78.406,169.260,36.190,156.815
C03166=1041.312,-36.306,-78.419,169.262,36.190,156.815
C03167=1041.318,-36.056,-78.431,169.264,36.191,156.815
C03168=1041.324,-35.775,-78.447,169.266,36.192,156.815
C03169=1041.331,-35.495,-78.461,169.269,36.192,156.815
C03170=1041.338,-35.213,-78.477,169.271,36.193,156.815
C03171=1041.345,-34.932,-78.491,169.273,36.194,156.815
C03172=1041.352,-34.683,-78.505,169.276,36.195,156.815
C03173=1041.358,-34.433,-78.518,169.278,36.195,156.815
C03174=1041.365,-34.183,-78.532,169.280,36.196,156.816
C03175=1041.371,-33.934,-78.545,169.282,36.196,156.816
C03176=1041.377,-33.684,-78.557,169.285,36.197,156.816
C03177=1041.383,-33.435,-78.571,169.287,36.198,156.816
C03178=1041.390,-33.185,-78.584,169.289,36.198,156.816
C03179=1041.395,-32.936,-78.598,169.292,36.199,156.816
C03180=1041.402,-32.686,-78.611,169.294,36.200,156.816
C03181=1041.408,-32.436,-78.625,169.296,36.200,156.816
C03182=1041.415,-32.187,-78.638,169.298,36.201,156.816
C03183=1041.421,-31.938,-78.652,169.300,36.202,156.817
C03184=1041.427,-31.689,-78.665,169.302,36.202,156.817
C03185=1041.434,-31.438,-78.678,169.304,36.203,156.817
C03186=1041.440,-31.189,-78.691,169.306,36.204,156.817
C03187=1041.446,-30.939,-78.704,169.309,36.204,156.817
C03188=1041.453,-30.689,-78.718,169.311,36.205,156.817
C03189=1041.459,-30.440,-78.731,169.313,36.206,156.817
C03190=1041.464,-30.191,-78.745,169.315,36.206,156.817
C03191=1041.471,-29.941,-78.759,169.317,36.207,156.817
C03192=1041.477,-29.691,-78.772,169.319,36.208,156.818
C03193=1041.484,-29.442,-78.785,169.322,36.208,156.818
C03194=1041.491,-29.192,-78.799,169.324,36.209,156.818
C03195=1041.497,-28.943,-78.812,169.327,36.210,156.818
C03196=1041.504,-28.693,-78.826,169.329,36.210,156.818
C03197=1041.510,-28.444,-78.839,169.331,36.211,156.818
C03198=1041.516,-28.194,-78.852,169.333,36.212,156.818
C03199=1041.523,-27.944,-78.866,169.335,36.212,156.818
C03200=1041.528,-27.695,-78.880,169.337,36.213,156.818
C03201=1041.535,-27.445,-78.894,169.339,36.213,156.819
C03202=1041.541,-27.196,-78.907,169.341,36.214,156.819
C03203=1041.548,-26.946,-78.920,169.343,36.215,156.819
C03204=1041.555,-26.697,-78.934,169.346,36.215,156.819
C03205=1041.560,-26.447,-78.948,169.348,36.216,156.819
C03206=1041.566,-26.198,-78.962,169.350,36.217,156.819
C03207=1041.573,-25.948,-78.975,169.352,36.217,156.819
C03208=1041.579,-25.699,-78.989,169.354,36.218,156.819
C03209=1041.585,-25.449,-79.003,169.357,36.219,156.820
C03210=1041.592,-25.199,-79.016,169.359,36.220,156.820
C03211=1041.597,-24.950,-79.031,169.361,36.221,156.820
C03212=1041.604,-24.700,-79.044,169.363,36.221,156.820
C03213=1041.610,-24.451,-79.058,169.365,36.222,156.820
C03214=1041.617,-24.201,-79.072,169.367,36.223,156.820
C03215=1041.623,-23.952,-79.085,169.369,36.224,156.820
C03216=1041.629,-23.703,-79.100,169.371,36.225,156.820
C03217=1041.635,-23.453,-79.113,169.373,36.225,156.821
C03218=1041.642,-23.203,-79.126,169.375,36.226,156.821
C03219=1041.648,-22.953,-79.141,169.378,36.227,156.821
C03220=1041.654,-22.704,-79.154,169.380,36.227,156.821
C03221=1041.660,-22.454,-79.169,169.382,36.228,156.821
C03222=1041.666,-22.205,-79.182,169.384,36.229,156.821
C03223=1041.673,-21.955,-79.196,169.387,36.230,156.821
C03224=1041.679,-21.706,-79.210,169.389,36.230,156.821
C03225=1041.685,-21.457,-79.224,169.391,36.231,156.822
C03226=1041.692,-21.207,-79.237,169.393,36.232,156.822
C03227=1041.698,-20.957,-79.251,169.395,36.232,156.822
C03228=1041.705,-20.708,-79.266,169.397,36.233,156.822
C03229=1041.710,-20.458,-79.279,169.399,36.234,156.822
C03230=1041.717,-20.208,-79.293,169.401,36.235,156.822
C03231=1041.723,-19.960,-79.307,169.403,36.236,156.822
C03232=1041.731,-19.677,-79.322,169.406,36.236,156.822
C03233=1041.738,-19.396,-79.338,169.408,36.238,156.823
C03234=1041.744,-19.114,-79.355,169.410,36.238,156.823
C03235=1041.752,-18.832,-79.370,169.412,36.239,156.823
C03236=1041.759,-18.582,-79.385,169.415,36.240,156.823
C03237=1041.765,-18.333,-79.398,169.418,36.240,156.823
C03238=1041.771,-18.083,-79.412,169.420,36.242,156.823
C03239=1041.778,-17.834,-79.426,169.422,36.242,156.823
C03240=1041.784,-17.584,-79.440,169.424,36.243,156.824
C03241=1041.790,-17.335,-79.454,169.426,36.244,156.824
C03242=1041.796,-17.085,-79.468,169.428,36.244,156.824
C03243=1041.802,-16.836,-79.482,169.430,36.245,156.824
C03244=1041.810,-16.586,-79.496,169.432,36.246,156.824
C03245=1041.816,-16.336,-79.510,169.434,36.247,156.824
C03246=1041.822,-16.087,-79.524,169.436,36.247,156.824
C03247=1041.828,-15.837,-79.539,169.438,36.248,156.825
C03248=1041.835,-15.588,-79.553,169.440,36.249,156.825
C03249=1041.841,-15.338,-79.567,169.442,36.249,156.825
C03250=1041.847,-15.090,-79.581,169.445,36.251,156.825
C03251=1041.853,-14.839,-79.595,169.447,36.251,156.825
C03252=1041.861,-14.590,-79.609,169.449,36.252,156.825
C03253=1041.866,-14.340,-79.623,169.451,36.253,156.825
C03254=1041.872,-14.091,-79.638,169.453,36.254,156.826
C03255=1041.879,-13.841,-79.651,169.455,36.255,156.826
C03256=1041.885,-13.592,-79.666,169.457,36.256,156.826
C03257=1041.891,-13.342,-79.680,169.459,36.257,156.826
C03258=1041.898,-13.093,-79.695,169.461,36.257,156.826
C03259=1041.904,-12.843,-79.710,169.463,36.258,156.826
C03260=1041.909,-12.594,-79.723,169.465,36.259,156.826
C03261=1041.917,-12.344,-79.738,169.467,36.260,156.827
C03262=1041.922,-12.095,-79.752,169.469,36.260,156.827
C03263=1041.928,-11.845,-79.767,169.472,36.262,156.827
C03264=1041.936,-11.596,-79.781,169.474,36.262,156.827
C03265=1041.941,-11.346,-79.795,169.476,36.263,156.827
C03266=1041.947,-11.096,-79.810,169.478,36.264,156.827
C03267=1041.955,-10.847,-79.824,169.480,36.265,156.827
C03268=1041.960,-10.598,-79.838,169.482,36.266,156.828
C03269=1041.966,-10.348,-79.853,169.484,36.267,156.828
C03270=1041.973,-10.099,-79.867,169.486,36.268,156.828
C03271=1041.979,-9.849,-79.881,169.488,36.268,156.828
C03272=1041.985,-9.599,-79.896,169.490,36.269,156.828
C03273=1041.991,-9.350,-79.911,169.492,36.270,156.828
C03274=1041.998,-9.101,-79.925,169.494,36.271,156.828
C03275=1042.004,-8.851,-79.939,169.497,36.271,156.829
C03276=1042.010,-8.602,-79.954,169.499,36.273,156.829
C03277=1042.017,-8.352,-79.968,169.501,36.273,156.829
C03278=1042.024,-8.103,-79.983,169.503,36.274,156.829
C03279=1042.030,-7.852,-79.997,169.505,36.275,156.829
C03280=1042.036,-7.604,-80.011,169.507,36.276,156.829
C03281=1042.043,-7.354,-80.026,169.509,36.277,156.829
C03282=1042.049,-7.105,-80.041,169.511,36.278,156.830
C03283=1042.055,-6.855,-80.055,169.513,36.279,156.830
C03284=1042.062,-6.606,-80.069,169.515,36.279,156.830
C03285=1042.068,-6.356,-80.084,169.517,36.281,156.830
C03286=1042.074,-6.106,-80.099,169.519,36.281,156.830
C03287=1042.081,-5.858,-80.113,169.521,36.282,156.830
C03288=1042.087,-5.607,-80.128,169.523,36.282,156.831
C03289=1042.093,-5.358,-80.142,169.525,36.284,156.831
C03290=1042.099,-5.109,-80.157,169.527,36.284,156.831
C03291=1042.106,-4.859,-80.171,169.529,36.285,156.831
C03292=1042.113,-4.610,-80.186,169.531,36.286,156.831
C03293=1042.119,-4.360,-80.201,169.533,36.287,156.831
C03294=1042.126,-4.111,-80.216,169.535,36.288,156.831
C03295=1042.132,-3.861,-80.229,169.537,36.289,156.832
C03296=1042.139,-3.578,-80.247,169.539,36.290,156.832
C03297=1042.147,-3.294,-80.263,169.542,36.291,156.832
C03298=1042.153,-3.010,-80.280,169.545,36.292,156.832
C03299=1042.160,-2.728,-80.297,169.547,36.293,156.832
C03300=1042.167,-2.478,-80.312,169.549,36.294,156.833
C03301=1042.173,-2.229,-80.327,169.551,36.295,156.833
C03302=1042.179,-1.979,-80.342,169.553,36.296,156.833
C03303=1042.185,-1.730,-80.357,169.555,36.297,156.833
C03304=1042.192,-1.480,-80.372,169.557,36.298,156.833
C03305=1042.198,-1.231,-80.386,169.558,36.299,156.833
C03306=1042.204,-0.981,-80.401,169.560,36.300,156.834
C03307=1042.210,-0.732,-80.416,169.562,36.301,156.834
C03308=1042.217,-0.482,-80.431,169.565,36.302,156.834
C03309=1042.222,-0.233,-80.446,169.567,36.302,156.834
C03310=1042.229,0.017,-80.461,169.569,36.304,156.834
C03311=1042.234,0.267,-80.476,169.571,36.304,156.834
C03312=1042.241,0.516,-80.491,169.573,36.306,156.835
C03313=1042.247,0.765,-80.506,169.575,36.306,156.835
C03314=1042.253,1.015,-80.521,169.577,36.308,156.835
C03315=1042.259,1.265,-80.536,169.579,36.308,156.835
C03316=1042.266,1.514,-80.551,169.581,36.310,156.835
C03317=1042.272,1.763,-80.566,169.582,36.310,156.835
C03318=1042.278,2.012,-80.581,169.585,36.311,156.836
C03319=1042.285,2.262,-80.596,169.587,36.312,156.836
C03320=1042.291,2.511,-80.611,169.589,36.313,156.836
C03321=1042.297,2.761,-80.626,169.591,36.314,156.836
C03322=1042.304,3.011,-80.641,169.593,36.315,156.836
C03323=1042.310,3.260,-80.655,169.595,36.316,156.836
C03324=1042.316,3.509,-80.671,169.597,36.317,156.837
C03325=1042.323,3.758,-80.686,169.599,36.318,156.837
C03326=1042.329,4.008,-80.701,169.601,36.319,156.837
C03327=1042.335,4.258,-80.716,169.602,36.320,156.837
C03328=1042.341,4.508,-80.731,169.604,36.321,156.837
C03329=1042.348,4.757,-80.747,169.607,36.322,156.837
C03330=1042.354,5.006,-80.762,169.609,36.323,156.838
C03331=1042.361,5.256,-80.777,169.611,36.324,156.838
C03332=1042.366,5.505,-80.791,169.613,36.325,156.838
C03333=1042.373,5.755,-80.806,169.615,36.326,156.838
C03334=1042.379,6.004,-80.822,169.617,36.327,156.838
C03335=1042.386,6.253,-80.837,169.619,36.328,156.839
C03336=1042.392,6.503,-80.852,169.620,36.329,156.839
C03337=1042.399,6.753,-80.867,169.622,36.329,156.839
C03338=1042.404,7.002,-80.883,169.624,36.331,156.839
C03339=1042.411,7.252,-80.898,169.627,36.331,156.839
C03340=1042.417,7.501,-80.913,169.629,36.333,156.839
C03341=1042.424,7.750,-80.929,169.631,36.333,156.840
C03342=1042.430,8.000,-80.943,169.633,36.335,156.840
C03343=1042.436,8.249,-80.958,169.635,36.335,156.840
C03344=1042.442,8.499,-80.973,169.637,36.337,156.840
C03345=1042.449,8.748,-80.989,169.638,36.337,156.840
C03346=1042.456,8.997,-81.004,169.640,36.338,156.840
C03347=1042.461,9.247,-81.019,169.642,36.339,156.841
C03348=1042.468,9.496,-81.035,169.644,36.340,156.841
C03349=1042.474,9.746,-81.050,169.646,36.341,156.841
C03350=1042.481,9.995,-81.065,169.649,36.342,156.841
C03351=1042.487,10.245,-81.080,169.651,36.343,156.841
C03352=1042.494,10.494,-81.095,169.653,36.344,156.842
C03353=1042.500,10.743,-81.111,169.655,36.345,156.842
C03354=1042.507,10.993,-81.126,169.656,36.346,156.842
C03355=1042.513,11.243,-81.141,169.658,36.347,156.842
C03356=1042.519,11.492,-81.157,169.660,36.347,156.842
C03357=1042.526,11.742,-81.172,169.662,36.349,156.842
C03358=1042.532,11.991,-81.188,169.664,36.349,156.842
C03359=1042.539,12.240,-81.203,169.666,36.351,156.843
C03360=1042.546,12.526,-81.220,169.669,36.352,156.843
C03361=1042.554,12.811,-81.238,169.671,36.353,156.843
C03362=1042.561,13.096,-81.256,169.673,36.354,156.843
C03363=1042.568,13.382,-81.273,169.675,36.355,156.843
C03364=1042.574,13.631,-81.289,169.677,36.356,156.844
C03365=1042.581,13.881,-81.304,169.679,36.357,156.844
C03366=1042.587,14.130,-81.320,169.681,36.358,156.844
C03367=1042.594,14.380,-81.335,169.683,36.359,156.844
C03368=1042.600,14.629,-81.351,169.685,36.360,156.844
C03369=1042.606,14.879,-81.366,169.688,36.361,156.844
C03370=1042.613,15.128,-81.381,169.689,36.362,156.845
C03371=1042.619,15.377,-81.398,169.691,36.363,156.845
C03372=1042.625,15.627,-81.413,169.693,36.364,156.845
C03373=1042.631,15.876,-81.429,169.695,36.365,156.845
C03374=1042.638,16.126,-81.444,169.697,36.366,156.845
C03375=1042.644,16.375,-81.459,169.699,36.367,156.846
C03376=1042.650,16.624,-81.476,169.700,36.368,156.846
C03377=1042.657,16.874,-81.491,169.702,36.369,156.846
C03378=1042.663,17.123,-81.507,169.705,36.370,156.846
C03379=1042.669,17.373,-81.522,169.707,36.371,156.846
C03380=1042.676,17.622,-81.538,169.709,36.372,156.847
C03381=1042.682,17.872,-81.554,169.711,36.373,156.847
C03382=1042.689,18.121,-81.569,169.712,36.374,156.847
C03383=1042.694,18.371,-81.585,169.714,36.376,156.847
C03384=1042.701,18.620,-81.601,169.716,36.376,156.847
C03385=1042.708,18.869,-81.616,169.718,36.377,156.848
C03386=1042.713,19.119,-81.632,169.720,36.378,156.848
C03387=1042.720,19.368,-81.648,169.722,36.379,156.848
C03388=1042.726,19.617,-81.664,169.724,36.381,156.848
C03389=1042.733,19.867,-81.679,169.726,36.381,156.848
C03390=1042.739,20.116,-81.695,169.728,36.383,156.848
C03391=1042.746,20.366,-81.711,169.730,36.384,156.849
C03392=1042.751,20.616,-81.727,169.732,36.384,156.849
C03393=1042.758,20.865,-81.743,169.733,36.386,156.849
C03394=1042.764,21.114,-81.759,169.735,36.387,156.849
C03395=1042.771,21.363,-81.774,169.737,36.388,156.849
C03396=1042.777,21.613,-81.791,169.739,36.389,156.850
C03397=1042.783,21.862,-81.806,169.742,36.390,156.850
C03398=1042.789,22.112,-81.822,169.744,36.391,156.850
C03399=1042.796,22.361,-81.838,169.745,36.392,156.850
C03400=1042.802,22.611,-81.854,169.747,36.393,156.850
C03401=1042.809,22.860,-81.870,169.749,36.394,156.851
C03402=1042.815,23.110,-81.885,169.751,36.395,156.851
C03403=1042.821,23.359,-81.902,169.753,36.397,156.851
C03404=1042.827,23.608,-81.917,169.754,36.397,156.851
C03405=1042.833,23.858,-81.934,169.756,36.399,156.851
C03406=1042.840,24.107,-81.949,169.759,36.400,156.852
C03407=1042.846,24.357,-81.966,169.761,36.400,156.852
C03408=1042.853,24.606,-81.982,169.763,36.402,156.852
C03409=1042.859,24.856,-81.997,169.764,36.403,156.852
C03410=1042.865,25.105,-82.013,169.766,36.404,156.852
C03411=1042.871,25.354,-82.029,169.768,36.405,156.852
C03412=1042.878,25.604,-82.046,169.770,36.406,156.853
C03413=1042.885,25.853,-82.061,169.772,36.407,156.853
C03414=1042.891,26.102,-82.078,169.773,36.408,156.853
C03415=1042.897,26.351,-82.093,169.776,36.409,156.853
C03416=1042.903,26.601,-82.109,169.778,36.410,156.853
C03417=1042.910,26.851,-82.126,169.780,36.411,156.854
C03418=1042.916,27.100,-82.142,169.782,36.413,156.854
C03419=1042.922,27.349,-82.158,169.783,36.413,156.854
C03420=1042.929,27.598,-82.174,169.785,36.414,156.854
C03421=1042.935,27.848,-82.190,169.787,36.416,156.854
C03422=1042.942,28.098,-82.207,169.789,36.417,156.855
C03423=1042.948,28.347,-82.222,169.791,36.418,156.855
C03424=1042.955,28.634,-82.241,169.794,36.419,156.855
C03425=1042.962,28.920,-82.259,169.796,36.420,156.855
C03426=1042.969,29.206,-82.278,169.798,36.421,156.856
C03427=1042.977,29.493,-82.296,169.800,36.423,156.856
C03428=1042.983,29.743,-82.313,169.802,36.424,156.856
C03429=1042.989,29.992,-82.330,169.803,36.425,156.856
C03430=1042.995,30.241,-82.346,169.805,36.427,156.856
C03431=1043.001,30.491,-82.362,169.808,36.427,156.857
C03432=1043.009,30.741,-82.378,169.810,36.428,156.857
C03433=1043.014,30.990,-82.394,169.811,36.430,156.857
C03434=1043.020,31.239,-82.411,169.813,36.431,156.857
C03435=1043.026,31.489,-82.427,169.815,36.432,156.857
C03436=1043.033,31.739,-82.443,169.817,36.433,156.858
C03437=1043.040,31.987,-82.460,169.818,36.434,156.858
C03438=1043.046,32.236,-82.476,169.820,36.435,156.858
C03439=1043.052,32.486,-82.492,169.822,36.436,156.858
C03440=1043.058,32.736,-82.509,169.825,36.437,156.858
C03441=1043.064,32.985,-82.525,169.827,36.439,156.859
C03442=1043.071,33.234,-82.541,169.828,36.440,156.859
C03443=1043.077,33.484,-82.557,169.830,36.440,156.859
C03444=1043.084,33.733,-82.574,169.832,36.442,156.859
C03445=1043.090,33.982,-82.591,169.834,36.443,156.859
C03446=1043.096,34.232,-82.607,169.835,36.444,156.860
C03447=1043.102,34.482,-82.624,169.837,36.445,156.860
C03448=1043.109,34.731,-82.639,169.840,36.446,156.860
C03449=1043.115,34.979,-82.656,169.842,36.447,156.860
C03450=1043.122,35.230,-82.673,169.843,36.449,156.861
C03451=1043.128,35.479,-82.689,169.845,36.449,156.861
C03452=1043.134,35.728,-82.705,169.847,36.451,156.861
C03453=1043.141,35.978,-82.723,169.849,36.452,156.861
C03454=1043.147,36.227,-82.738,169.851,36.453,156.861
C03455=1043.153,36.476,-82.755,169.852,36.454,156.861
C03456=1043.160,36.725,-82.772,169.855,36.455,156.862
C03457=1043.166,36.975,-82.788,169.857,36.456,156.862
C03458=1043.172,37.224,-82.804,169.859,36.458,156.862
C03459=1043.179,37.474,-82.821,169.860,36.458,156.862
C03460=1043.185,37.723,-82.838,169.862,36.459,156.863
C03461=1043.191,37.972,-82.854,169.864,36.461,156.863
C03462=1043.197,38.222,-82.871,169.866,36.462,156.863
C03463=1043.204,38.471,-82.888,169.867,36.463,156.863
C03464=1043.209,38.720,-82.904,169.870,36.465,156.863
C03465=1043.216,38.970,-82.921,169.872,36.465,156.864
C03466=1043.222,39.219,-82.938,169.874,36.466,156.864
C03467=1043.228,39.469,-82.954,169.875,36.468,156.864
C03468=1043.235,39.718,-82.971,169.877,36.469,156.864
C03469=1043.241,39.967,-82.988,169.879,36.470,156.865
C03470=1043.248,40.217,-83.005,169.881,36.472,156.865
C03471=1043.254,40.466,-83.021,169.882,36.472,156.865
C03472=1043.260,40.715,-83.037,169.885,36.473,156.865
C03473=1043.267,40.965,-83.055,169.887,36.475,156.865
C03474=1043.273,41.214,-83.071,169.888,36.476,156.866
C03475=1043.279,41.463,-83.088,169.890,36.477,156.866
C03476=1043.285,41.713,-83.105,169.892,36.478,156.866
C03477=1043.292,41.962,-83.122,169.894,36.479,156.866
C03478=1043.297,42.212,-83.139,169.895,36.480,156.866
C03479=1043.304,42.461,-83.156,169.897,36.482,156.867
C03480=1043.310,42.710,-83.172,169.900,36.483,156.867
C03481=1043.317,42.960,-83.189,169.902,36.484,156.867
C03482=1043.323,43.209,-83.206,169.903,36.485,156.867
C03483=1043.329,43.458,-83.223,169.905,36.486,156.867
C03484=1043.335,43.708,-83.239,169.907,36.487,156.868
C03485=1043.341,43.957,-83.257,169.909,36.489,156.868
C03486=1043.347,44.207,-83.273,169.910,36.490,156.868
C03487=1043.354,44.456,-83.290,169.912,36.491,156.868
C03488=1043.361,44.743,-83.310,169.915,36.493,156.869
C03489=1043.368,45.029,-83.330,169.917,36.494,156.869
C03490=1043.375,45.315,-83.349,169.919,36.496,156.869
C03491=1043.382,45.602,-83.370,169.921,36.497,156.869
C03492=1043.388,45.851,-83.386,169.922,36.498,156.870
C03493=1043.394,46.100,-83.403,169.924,36.499,156.870
C03494=1043.400,46.350,-83.420,169.927,36.501,156.870
C03495=1043.406,46.599,-83.437,169.929,36.502,156.870
C03496=1043.413,46.849,-83.454,169.930,36.503,156.871
C03497=1043.418,47.098,-83.471,169.932,36.504,156.871
C03498=1043.425,47.348,-83.489,169.934,36.506,156.871
C03499=1043.432,47.596,-83.505,169.935,36.507,156.871
C03500=1043.437,47.845,-83.523,169.937,36.508,156.872
C03501=1043.444,48.095,-83.540,169.939,36.509,156.872
C03502=1043.450,48.344,-83.557,169.942,36.511,156.872
C03503=1043.456,48.594,-83.575,169.943,36.512,156.872
C03504=1043.462,48.843,-83.591,169.945,36.513,156.873
C03505=1043.469,49.093,-83.608,169.947,36.514,156.873
C03506=1043.474,49.342,-83.626,169.948,36.516,156.873
C03507=1043.481,49.591,-83.643,169.950,36.516,156.873
C03508=1043.487,49.840,-83.659,169.952,36.518,156.873
C03509=1043.493,50.090,-83.677,169.955,36.519,156.874
C03510=1043.500,50.339,-83.694,169.956,36.520,156.874
C03511=1043.506,50.588,-83.712,169.958,36.521,156.874
C03512=1043.512,50.838,-83.728,169.960,36.523,156.874
C03513=1043.518,51.087,-83.746,169.961,36.524,156.875
C03514=1043.525,51.336,-83.763,169.963,36.525,156.875
C03515=1043.531,51.586,-83.781,169.965,36.526,156.875
C03516=1043.537,51.835,-83.798,169.968,36.528,156.875
C03517=1043.543,52.085,-83.815,169.969,36.529,156.875
C03518=1043.549,52.334,-83.832,169.971,36.530,156.876
C03519=1043.556,52.583,-83.849,169.973,36.531,156.876
C03520=1043.562,52.832,-83.867,169.974,36.532,156.876
C03521=1043.568,53.082,-83.884,169.976,36.533,156.876
C03522=1043.575,53.331,-83.901,169.978,36.535,156.877
C03523=1043.580,53.581,-83.918,169.979,36.536,156.877
C03524=1043.587,53.830,-83.936,169.982,36.537,156.877
C03525=1043.594,54.079,-83.953,169.984,36.538,156.877
C03526=1043.600,54.329,-83.971,169.986,36.540,156.877
C03527=1043.606,54.577,-83.987,169.987,36.541,156.878
C03528=1043.612,54.827,-84.005,169.989,36.542,156.878
C03529=1043.619,55.077,-84.023,169.991,36.543,156.878
C03530=1043.625,55.325,-84.040,169.992,36.544,156.878
C03531=1043.631,55.575,-84.058,169.995,36.545,156.879
C03532=1043.638,55.824,-84.075,169.997,36.547,156.879
C03533=1043.644,56.074,-84.093,169.999,36.548,156.879
C03534=1043.650,56.324,-84.109,170.000,36.549,156.879
C03535=1043.656,56.572,-84.126,170.002,36.550,156.880
C03536=1043.663,56.822,-84.144,170.004,36.552,156.880
C03537=1043.669,57.071,-84.161,170.005,36.553,156.880
C03538=1043.676,57.320,-84.178,170.008,36.554,156.880
C03539=1043.682,57.570,-84.196,170.010,36.555,156.880
C03540=1043.688,57.819,-84.213,170.012,36.556,156.881
C03541=1043.694,58.068,-84.231,170.013,36.557,156.881
C03542=1043.701,58.318,-84.249,170.015,36.559,156.881
C03543=1043.707,58.567,-84.266,170.017,36.560,156.881
C03544=1043.713,58.816,-84.283,170.018,36.561,156.882
C03545=1043.720,59.066,-84.301,170.020,36.562,156.882
C03546=1043.726,59.315,-84.318,170.023,36.564,156.882
C03547=1043.733,59.564,-84.336,170.025,36.564,156.882
C03548=1043.739,59.814,-84.354,170.026,36.565,156.882
C03549=1043.745,60.063,-84.371,170.028,36.567,156.883
C03550=1043.752,60.311,-84.389,170.030,36.568,156.883
C03551=1043.758,60.561,-84.407,170.031,36.569,156.883
C03552=1043.765,60.847,-84.427,170.033,36.570,156.883
C03553=1043.773,61.134,-84.447,170.036,36.572,156.884
C03554=1043.780,61.420,-84.467,170.038,36.573,156.884
C03555=1043.788,61.706,-84.487,170.040,36.574,156.884
C03556=1043.794,61.955,-84.504,170.042,36.575,156.884
C03557=1043.801,62.205,-84.521,170.044,36.577,156.884
C03558=1043.807,62.454,-84.539,170.046,36.578,156.885
C03559=1043.814,62.704,-84.557,170.047,36.579,156.885
C03560=1043.819,62.952,-84.575,170.050,36.580,156.885
C03561=1043.826,63.202,-84.592,170.052,36.581,156.885
C03562=1043.833,63.451,-84.610,170.053,36.582,156.886
C03563=1043.839,63.701,-84.628,170.055,36.584,156.886
C03564=1043.845,63.949,-84.645,170.057,36.585,156.886
C03565=1043.852,64.199,-84.663,170.059,36.586,156.886
C03566=1043.858,64.448,-84.681,170.060,36.587,156.887
C03567=1043.865,64.698,-84.699,170.062,36.589,156.887
C03568=1043.870,64.947,-84.716,170.065,36.590,156.887
C03569=1043.876,65.197,-84.734,170.066,36.591,156.887
C03570=1043.883,65.446,-84.753,170.068,36.592,156.887
C03571=1043.889,65.694,-84.770,170.070,36.594,156.888
C03572=1043.895,65.944,-84.788,170.071,36.595,156.888
C03573=1043.901,66.194,-84.806,170.073,36.596,156.888
C03574=1043.909,66.443,-84.824,170.075,36.597,156.888
C03575=1043.914,66.692,-84.841,170.077,36.599,156.889
C03576=1043.920,66.941,-84.859,170.079,36.600,156.889
C03577=1043.927,67.190,-84.877,170.081,36.601,156.889
C03578=1043.933,67.440,-84.895,170.083,36.602,156.889
C03579=1043.939,67.689,-84.913,170.084,36.604,156.890
C03580=1043.945,67.938,-84.931,170.086,36.605,156.890
C03581=1043.952,68.188,-84.949,170.089,36.606,156.890
C03582=1043.958,68.437,-84.967,170.090,36.607,156.890
C03583=1043.964,68.686,-84.985,170.092,36.609,156.891
C03584=1043.970,68.936,-85.003,170.094,36.610,156.891
C03585=1043.977,69.185,-85.020,170.095,36.611,156.891
C03586=1043.984,69.434,-85.039,170.097,36.612,156.891
C03587=1043.989,69.683,-85.056,170.099,36.614,156.892
C03588=1043.996,69.932,-85.075,170.101,36.615,156.892
C03589=1044.002,70.182,-85.093,170.103,36.616,156.892
C03590=1044.008,70.431,-85.112,170.105,36.617,156.892
C03591=1044.014,70.681,-85.129,170.106,36.619,156.892
C03592=1044.020,70.930,-85.147,170.108,36.620,156.893
C03593=1044.027,71.179,-85.165,170.110,36.621,156.893
C03594=1044.033,71.428,-85.183,170.112,36.622,156.893
C03595=1044.039,71.678,-85.202,170.114,36.624,156.893
C03596=1044.045,71.927,-85.219,170.116,36.625,156.894
C03597=1044.051,72.176,-85.238,170.118,36.626,156.894
C03598=1044.058,72.425,-85.256,170.119,36.627,156.894
C03599=1044.064,72.675,-85.274,170.121,36.629,156.894
C03600=1044.070,72.924,-85.292,170.123,36.630,156.895
C03601=1044.076,73.173,-85.311,170.124,36.631,156.895
C03602=1044.082,73.422,-85.329,170.127,36.632,156.895
C03603=1044.089,73.671,-85.347,170.129,36.634,156.895
C03604=1044.096,73.920,-85.365,170.130,36.635,156.896
C03605=1044.102,74.170,-85.383,170.132,36.636,156.896
C03606=1044.108,74.419,-85.402,170.134,36.637,156.896
C03607=1044.114,74.668,-85.419,170.135,36.639,156.896
C03608=1044.120,74.917,-85.438,170.137,36.640,156.897
C03609=1044.126,75.167,-85.456,170.140,36.641,156.897
C03610=1044.133,75.416,-85.475,170.141,36.643,156.897
C03611=1044.139,75.665,-85.493,170.143,36.644,156.897
C03612=1044.145,75.915,-85.511,170.145,36.646,156.898
